(* IEC 61131-3 sources: RL_MAR/experiments/results/ablation/Ablation_no_role_config_deepseek-ai_DeepSeek-V3.2_20260603_074104, 94 files *)

(* ---- hard_92.st ---- *)
FUNCTION_BLOCK FB_BreakerControlSystem
VAR_INPUT
    B10_1_Trip : BOOL;
    B10_1_Close : BOOL;
    B10_2_Trip : BOOL;
    B10_2_Close : BOOL;
    B10_12_Trip : BOOL;
    B10_12_Close : BOOL;
    B54_Trip : BOOL;
    B54_Close : BOOL;
    B55_Trip : BOOL;
    B55_Close : BOOL;
    B56_Trip : BOOL;
    B56_Close : BOOL;
    B57_Trip : BOOL;
    B57_Close : BOOL;
END_VAR

VAR_OUTPUT
    Point_1a : INT;
    Point_2a : INT;
    Point_3a : INT;
    Point_4a : INT;
    B10_1_Opened : BOOL;
    B10_1_Closed : BOOL;
    B10_2_Opened : BOOL;
    B10_2_Closed : BOOL;
    B10_12_Opened : BOOL;
    B10_12_Closed : BOOL;
    B54_Opened : BOOL;
    B54_Closed : BOOL;
    B55_Opened : BOOL;
    B55_Closed : BOOL;
    B56_Opened : BOOL;
    B56_Closed : BOOL;
    B57_Opened : BOOL;
    B57_Closed : BOOL;
END_VAR

VAR
    SEL86_OUT : INT;
    MOVE89_OUT : INT;
    SEL66_OUT : INT;
    MOVE69_OUT : INT;
    SEL96_OUT : INT;
    MOVE99_OUT : INT;
    SEL106_OUT : INT;
    MOVE109_OUT : INT;
END_VAR

// Breaker B10_1 State Transition
IF B10_1_Close THEN
    B10_1_Closed := TRUE;
    B10_1_Opened := FALSE;
ELSIF B10_1_Trip THEN
    B10_1_Closed := FALSE;
    B10_1_Opened := TRUE;
END_IF;

// Breaker B10_2 State Transition
IF B10_2_Close THEN
    B10_2_Closed := TRUE;
    B10_2_Opened := FALSE;
ELSIF B10_2_Trip THEN
    B10_2_Closed := FALSE;
    B10_2_Opened := TRUE;
END_IF;

// Breaker B10_12 State Transition
IF B10_12_Close THEN
    B10_12_Closed := TRUE;
    B10_12_Opened := FALSE;
ELSIF B10_12_Trip THEN
    B10_12_Closed := FALSE;
    B10_12_Opened := TRUE;
END_IF;

// Breaker B54 State Transition
IF B54_Close THEN
    B54_Closed := TRUE;
    B54_Opened := FALSE;
ELSIF B54_Trip THEN
    B54_Closed := FALSE;
    B54_Opened := TRUE;
END_IF;

// Breaker B55 State Transition
IF B55_Close THEN
    B55_Closed := TRUE;
    B55_Opened := FALSE;
ELSIF B55_Trip THEN
    B55_Closed := FALSE;
    B55_Opened := TRUE;
END_IF;

// Breaker B56 State Transition
IF B56_Close THEN
    B56_Closed := TRUE;
    B56_Opened := FALSE;
ELSIF B56_Trip THEN
    B56_Closed := FALSE;
    B56_Opened := TRUE;
END_IF;

// Breaker B57 State Transition
IF B57_Close THEN
    B57_Closed := TRUE;
    B57_Opened := FALSE;
ELSIF B57_Trip THEN
    B57_Closed := FALSE;
    B57_Opened := TRUE;
END_IF;

// Point_1a Calculation
IF B54_Closed AND ((B10_12_Closed AND B10_1_Closed) OR B10_2_Closed) THEN
    Point_1a := 0;
ELSE
    Point_1a := 138;
END_IF;

// Point_2a Calculation
IF B55_Closed AND ((B10_12_Closed AND B10_1_Closed) OR B10_2_Closed) THEN
    Point_2a := 0;
ELSE
    Point_2a := 138;
END_IF;

// Point_3a Calculation
IF B56_Closed AND ((B10_12_Closed AND B10_2_Closed) OR B10_1_Closed) THEN
    Point_3a := 0;
ELSE
    Point_3a := 138;
END_IF;

// Point_4a Calculation
IF B57_Closed AND ((B10_12_Closed AND B10_2_Closed) OR B10_1_Closed) THEN
    Point_4a := 0;
ELSE
    Point_4a := 138;
END_IF;

END_FUNCTION_BLOCK

(* ---- hard_93.st ---- *)
FUNCTION_BLOCK FB_CircuitControl
VAR_INPUT
    Reset_All_CB : BOOL;
    Current_Fault_on_TRSF1 : INT;
    Current_Fault_on_66BUS1 : INT;
END_VAR

VAR_OUTPUT
    Short_Circuit_TRSF1 : BOOL;
    Short_Circuit_66BUS : BOOL;
    Open_CB1_66KV : BOOL;
    Open_CB2_66KV : BOOL;
    Open_CB_TRSF1 : BOOL;
    Open_CB2_22KV : BOOL;
END_VAR

VAR
    Threshold500 : INT := 500;
    Prev_Open_CB2_22KV : BOOL;
    Prev_Open_CB1_66KV : BOOL;
    Prev_Open_CB_TRSF1 : BOOL;
    Temp_Open_CB2_22KV : BOOL;
    Temp_Open_CB1_66KV : BOOL;
    Temp_Open_CB_TRSF1 : BOOL;
END_VAR

(* Short circuit detection *)
Short_Circuit_66BUS := (Current_Fault_on_66BUS1 > Threshold500);
Short_Circuit_TRSF1 := (Current_Fault_on_TRSF1 > Threshold500);

(* Store previous states at the beginning of execution cycle *)
Prev_Open_CB2_22KV := Open_CB2_22KV;
Prev_Open_CB1_66KV := Open_CB1_66KV;
Prev_Open_CB_TRSF1 := Open_CB_TRSF1;

(* Initialize temporary variables with current output states *)
Temp_Open_CB2_22KV := Open_CB2_22KV;
Temp_Open_CB1_66KV := Open_CB1_66KV;
Temp_Open_CB_TRSF1 := Open_CB_TRSF1;

(* Reset handling - overrides all other logic *)
IF Reset_All_CB THEN
    Temp_Open_CB2_22KV := FALSE;
    Temp_Open_CB1_66KV := FALSE;
    Temp_Open_CB_TRSF1 := FALSE;
    Open_CB2_66KV := FALSE;  (* Even though spec says always TRUE, reset should override *)
ELSE
    (* First pass of circuit breaker control logic *)
    (* Open_CB2_22KV first condition *)
    IF (NOT Prev_Open_CB2_22KV) AND
       ((Open_CB1_66KV AND Open_CB_TRSF1) OR Short_Circuit_66BUS) THEN
        Temp_Open_CB2_22KV := TRUE;
    END_IF;

    (* Open_CB1_66KV first condition *)
    IF (NOT Temp_Open_CB2_22KV) AND
       ((Prev_Open_CB1_66KV AND Open_CB_TRSF1) OR Short_Circuit_66BUS) THEN
        Temp_Open_CB1_66KV := TRUE;
    END_IF;

    (* Open_CB_TRSF1 first condition *)
    IF (NOT Temp_Open_CB2_22KV) AND
       ((Open_CB1_66KV AND Prev_Open_CB_TRSF1) OR Short_Circuit_66BUS) THEN
        Temp_Open_CB_TRSF1 := TRUE;
    END_IF;

    (* Open_CB2_66KV always TRUE when not reset *)
    Open_CB2_66KV := TRUE;

    (* Update Open_CB2_22KV again *)
    IF (NOT Prev_Open_CB2_22KV) AND
       ((Open_CB2_66KV AND Temp_Open_CB1_66KV AND Temp_Open_CB_TRSF1) OR Short_Circuit_TRSF1) THEN
        Temp_Open_CB2_22KV := TRUE;
    END_IF;

    (* Update Open_CB1_66KV again *)
    IF (NOT Temp_Open_CB2_22KV) AND
       ((Open_CB2_66KV AND Prev_Open_CB1_66KV AND Temp_Open_CB_TRSF1) OR Short_Circuit_TRSF1) THEN
        Temp_Open_CB1_66KV := TRUE;
    END_IF;

    (* Update Open_CB_TRSF1 again *)
    IF (NOT Temp_Open_CB2_22KV) AND
       ((Open_CB2_66KV AND Temp_Open_CB1_66KV AND Prev_Open_CB_TRSF1) OR Short_Circuit_TRSF1) THEN
        Temp_Open_CB_TRSF1 := TRUE;
    END_IF;
END_IF;

(* Apply temporary states to outputs *)
Open_CB2_22KV := Temp_Open_CB2_22KV;
Open_CB1_66KV := Temp_Open_CB1_66KV;
Open_CB_TRSF1 := Temp_Open_CB_TRSF1;

END_FUNCTION_BLOCK

(* ---- hard_94.st ---- *)
FUNCTION_BLOCK FB_AdvancedCircuitBreakerControl
VAR_INPUT
    S_AL1_P_B1 : BOOL;
    S_AL1_P_B2 : BOOL;
    S_AL1_MCB : BOOL;
    MCB_BUSY : BOOL;
    MCB_ERROR : BOOL;
    S_AL1_MCBR : BOOL;
    MCBR_BUSY : BOOL;
    MCBR_ERROR : BOOL;
    S_AL1_P_B3 : BOOL;
    S_AL1_MCB2 : BOOL;
    S_AL1_MCBR2 : BOOL;
END_VAR

VAR_OUTPUT
    E_AL1_B1 : BOOL;
    PUWS_AL1_B1_PLUS : BOOL;
    PUWS_AL1_B1_RIGHT : BOOL;
    PAS_AL1_PLUS : BOOL;
    PAS_AL1_TURN : BOOL;
END_VAR

VAR
    PPAL1 : BOOL := 1;
    PP0 : BOOL := 1;
    PP1 : BOOL := 0;
    PP2 : BOOL := 0;
    PP3 : BOOL := 0;
    PP4 : BOOL := 0;
    MCB : BOOL := 1;
    PP5 : BOOL := 0;
    PP7 : BOOL := 0;
    PPL3 : BOOL := 0;
    PPL4 : BOOL := 0;
    MCBR : BOOL := 1;
    PPL5 : BOOL := 0;
    PPL7 : BOOL := 0;
    STABLE : BOOL := 0;
    MCB_CONTROL : BOOL;
END_VAR

METHOD MainLogic : BOOL
VAR_INPUT
END_VAR
VAR_OUTPUT
END_VAR
    STABLE := 0;

    WHILE (STABLE = 0) DO
        STABLE := 1;

        // PP0 to PP1
        IF PP0 AND (NOT MCB_CONTROL) AND (NOT PP1) THEN
            PP0 := 0;
            PP1 := 1;
            STABLE := 0;
        END_IF;

        // PP1 to PP2
        IF PP1 AND S_AL1_P_B1 AND (NOT PP2) THEN
            PP1 := 0;
            PP2 := 1;
            STABLE := 0;
        END_IF;

        // PP2 to PP3
        IF PP2 AND S_AL1_P_B2 AND (NOT MCB_CONTROL) AND (NOT PP3) THEN
            PP2 := 0;
            PP3 := 1;
            STABLE := 0;
        END_IF;

        // PP3 to PP4
        IF PP3 AND S_AL1_MCB AND (NOT PP4) AND (NOT PP1) THEN
            PP3 := 0;
            PP4 := 1;
            PP1 := 1;
            STABLE := 0;
        END_IF;

        // PP4 to PP5
        IF PP4 AND MCB AND MCB_BUSY AND (NOT PP5) THEN
            PP4 := 0;
            MCB := 0;
            PP5 := 1;
            STABLE := 0;
        END_IF;

        // PP5 to PP7
        IF PP5 AND S_AL1_MCB2 AND (NOT PP7) AND (NOT MCB) THEN
            PP5 := 0;
            PP7 := 1;
            MCB := 1;
            STABLE := 0;
        END_IF;

        // PP7 to End
        IF PP7 AND S_AL1_P_B3 THEN
            PP7 := 0;
            STABLE := 0;
        END_IF;

        // PP2 to PPL3
        IF PP2 AND S_AL1_P_B2 AND MCB_CONTROL AND (NOT PPL3) AND (NOT PP1) THEN
            PP2 := 0;
            PPL3 := 1;
            PP1 := 1;
            STABLE := 0;
        END_IF;

        // PPL3 to PPL4
        IF PPL3 AND S_AL1_MCBR AND (NOT PPL4) THEN
            PPL3 := 0;
            PPL4 := 1;
            STABLE := 0;
        END_IF;

        // PPL4 to PPL5
        IF PPL4 AND MCBR AND MCBR_BUSY AND (NOT PPL5) THEN
            PPL4 := 0;
            MCBR := 0;
            PPL5 := 1;
            STABLE := 0;
        END_IF;

        // PPL5 to PPL7
        IF PPL5 AND S_AL1_MCBR2 AND (NOT PPL7) AND (NOT MCBR) THEN
            PPL5 := 0;
            PPL7 := 1;
            MCBR := 1;
            STABLE := 0;
        END_IF;

        // PPL7 to End
        IF PPL7 AND S_AL1_P_B3 THEN
            PPL7 := 0;
            STABLE := 0;
        END_IF;
    END_WHILE;

    // Output Control Logic
    IF PP0 OR PP1 THEN
        E_AL1_B1 := 1;
    END_IF;

    IF PP3 THEN
        MCB_CONTROL := 1;
    END_IF;

    IF PPL3 OR PPL4 THEN
        PAS_AL1_PLUS := 1;
        PAS_AL1_TURN := 1;
    END_IF;

    IF PPAL1 OR PP2 THEN
        PUWS_AL1_B1_PLUS := 1;
    END_IF;

    IF PP2 OR PP3 OR PPL3 THEN
        E_AL1_B1 := 0;
    END_IF;

    IF PP0 OR PP3 THEN
        MCB_CONTROL := 0;
    END_IF;

    IF PP0 OR PP3 OR PP4 THEN
        PAS_AL1_PLUS := 0;
        PAS_AL1_TURN := 0;
    END_IF;

    IF PPAL1 OR PP2 THEN
        PUWS_AL1_B1_RIGHT := 0;
    END_IF;

    MainLogic := TRUE;
END_METHOD
END_FUNCTION_BLOCK

(* ---- hf_1.st ---- *)
FUNCTION_BLOCK StackMin
VAR_INPUT
    push : BOOL;
    pop : BOOL;
    reset : BOOL;
END_VAR
VAR_OUTPUT
    error : BOOL;
    status : WORD;
END_VAR
VAR_IN_OUT
    item : INT;
    stack : ARRAY[0..3] OF INT;
END_VAR
VAR
    top : INT := -1;
    i : INT;
    minIndex : INT;
    minValue : INT;
END_VAR

// Reset takes highest priority
IF reset THEN
    top := -1;
    error := FALSE;
    status := 16#0000;
ELSIF push THEN
    // Push operation
    IF top >= 3 THEN
        // Stack is full
        error := TRUE;
        status := 16#8A04;
    ELSE
        // Perform push
        top := top + 1;
        stack[top] := item;
        error := FALSE;
        status := 16#0000;
    END_IF;
ELSIF pop THEN
    // Pop operation (remove minimum value)
    IF top < 0 THEN
        // Stack is empty
        error := TRUE;
        status := 16#8A05;
    ELSE
        // Find minimum value and its index
        minIndex := 0;
        minValue := stack[0];
        FOR i := 1 TO top DO
            IF stack[i] < minValue THEN
                minValue := stack[i];
                minIndex := i;
            END_IF;
        END_FOR;

        // Return minimum value via item
        item := minValue;

        // Shift elements down to remove the minimum
        FOR i := minIndex TO top - 1 DO
            stack[i] := stack[i + 1];
        END_FOR;

        // Clear the last element (optional but clean)
        stack[top] := 0;

        // Update top index
        top := top - 1;

        error := FALSE;
        status := 16#0000;
    END_IF;
ELSE
    // No operation requested
    error := FALSE;
    status := 16#0000;
END_IF;

END_FUNCTION_BLOCK

(* ---- hf_10.st ---- *)
FUNCTION_BLOCK FloatingAverage
VAR_INPUT
    cyclicExecution : BOOL;
    trigger : BOOL;
    value : REAL;
    windowSize : INT;
    reset : BOOL;
END_VAR

VAR_OUTPUT
    average : REAL;
    windowSizeReached : BOOL;
    error : BOOL;
    status : WORD;
END_VAR

VAR
    dataBuffer : ARRAY[1..100] OF REAL; (* Buffer to store the data values *)
    bufferIndex : INT := 1; (* Index to track the current position in the buffer *)
    sum : REAL := 0.0; (* Sum of the data values in the buffer *)
    count : INT := 0; (* Number of valid data points in buffer *)
    triggerPrev : BOOL := FALSE; (* Previous trigger state for edge detection *)
END_VAR

(* Main execution logic *)
IF reset THEN
    (* Reset all internal variables *)
    bufferIndex := 1;
    sum := 0.0;
    count := 0;
    average := 0.0;
    windowSizeReached := FALSE;
    error := FALSE;
    status := 16#0000;

    (* Clear buffer *)
    FOR i := 1 TO 100 DO
        dataBuffer[i] := 0.0;
    END_FOR;

ELSIF windowSize < 1 OR windowSize > 100 THEN
    (* Window size error *)
    error := TRUE;
    status := 16#8200;
    windowSizeReached := FALSE;

ELSE
    (* Check if we should process new data *)
    IF cyclicExecution OR (trigger AND NOT triggerPrev) THEN
        (* Update buffer with new value *)
        dataBuffer[bufferIndex] := value;

        (* Update sum - subtract old value if buffer is full *)
        IF count < windowSize THEN
            sum := sum + value;
            count := count + 1;
        ELSE
            (* Calculate index of oldest value to be replaced *)
            VAR
                oldestIndex : INT;
            END_VAR

            oldestIndex := bufferIndex - windowSize + 1;
            IF oldestIndex < 1 THEN
                oldestIndex := oldestIndex + 100;
            END_IF;

            sum := sum - dataBuffer[oldestIndex] + value;
        END_IF;

        (* Update buffer index with circular buffer logic *)
        bufferIndex := bufferIndex + 1;
        IF bufferIndex > 100 THEN
            bufferIndex := 1;
        END_IF;

        (* Calculate average *)
        IF count > 0 THEN
            average := sum / count;
        ELSE
            average := 0.0;
        END_IF;

        (* Check if window size is reached *)
        windowSizeReached := (count >= windowSize);

        (* Clear error if window size is valid *)
        error := FALSE;
        status := 16#0000;
    END_IF;

    (* Update trigger previous state for edge detection *)
    triggerPrev := trigger;
END_IF;

END_FUNCTION_BLOCK

(* ---- hf_11.st ---- *)
FUNCTION_BLOCK FB_BottleProcessing
VAR_INPUT
    bottleSensor : BOOL;
    cleaningConfirmButton : BOOL;
    fillingConfirmButton : BOOL;
    cappingConfirmButton : BOOL;
    packingConfirmButton : BOOL;
    finishedButton : BOOL;
END_VAR

VAR_OUTPUT
    Pump_Motor : BOOL;
    Filling_Valve : BOOL;
    Capping_Machine : BOOL;
    Packing_Machine : BOOL;
    Completion_Light : BOOL;
END_VAR

VAR
    State : INT := 0; (* 0=Waiting, 1=Cleaning, 2=Filling, 3=Capping, 4=Packing, 5=Completed *)
END_VAR

CASE State OF
    0: (* Waiting *)
        (* State actions *)
        Pump_Motor := FALSE;
        Filling_Valve := FALSE;
        Capping_Machine := FALSE;
        Packing_Machine := FALSE;
        Completion_Light := FALSE;

        (* State transition *)
        IF bottleSensor THEN
            Pump_Motor := TRUE;
            State := 1;
        END_IF;

    1: (* Cleaning *)
        (* State actions *)
        Pump_Motor := TRUE;
        Filling_Valve := FALSE;
        Capping_Machine := FALSE;
        Packing_Machine := FALSE;
        Completion_Light := FALSE;

        (* State transition *)
        IF cleaningConfirmButton THEN
            Pump_Motor := FALSE;
            Filling_Valve := TRUE;
            State := 2;
        END_IF;

    2: (* Filling *)
        (* State actions *)
        Pump_Motor := FALSE;
        Filling_Valve := TRUE;
        Capping_Machine := FALSE;
        Packing_Machine := FALSE;
        Completion_Light := FALSE;

        (* State transition *)
        IF fillingConfirmButton THEN
            Filling_Valve := FALSE;
            Capping_Machine := TRUE;
            State := 3;
        END_IF;

    3: (* Capping *)
        (* State actions *)
        Pump_Motor := FALSE;
        Filling_Valve := FALSE;
        Capping_Machine := TRUE;
        Packing_Machine := FALSE;
        Completion_Light := FALSE;

        (* State transition *)
        IF cappingConfirmButton THEN
            Capping_Machine := FALSE;
            Packing_Machine := TRUE;
            State := 4;
        END_IF;

    4: (* Packing *)
        (* State actions *)
        Pump_Motor := FALSE;
        Filling_Valve := FALSE;
        Capping_Machine := FALSE;
        Packing_Machine := TRUE;
        Completion_Light := FALSE;

        (* State transition *)
        IF packingConfirmButton THEN
            Packing_Machine := FALSE;
            Completion_Light := TRUE;
            State := 5;
        END_IF;

    5: (* Completed *)
        (* State actions *)
        Pump_Motor := FALSE;
        Filling_Valve := FALSE;
        Capping_Machine := FALSE;
        Packing_Machine := FALSE;
        Completion_Light := TRUE;

        (* State transition *)
        IF finishedButton THEN
            Completion_Light := FALSE;
            (* All outputs already FALSE except Completion_Light which was just turned off *)
            State := 0;
        END_IF;

END_CASE;

END_FUNCTION_BLOCK

(* ---- hf_12.st ---- *)
FUNCTION_BLOCK MaterialMixing
VAR_INPUT
    estop : BOOL; (* Emergency Stop Signal, FALSE: Emergency stop triggered, TRUE: No emergency stop triggered *)
    opeMode : BOOL; (* Operation Mode, FALSE: Manual Operation Mode, TRUE: Automatic Operation Mode *)
    valveAStart : BOOL; (* Valve A Start Button *)
    valveBStart : BOOL; (* Valve B Start Button *)
    valveCStart : BOOL; (* Valve C Start Button *)
    valveDStart : BOOL; (* Valve D Start Button *)
    mixMotorStart : BOOL; (* Mixing Motor Start Button *)
    autoStart : BOOL; (* Automatic Start Button *)
    processMode : BOOL; (* Process Mode *)
    levelSensor : INT; (* Liquid Level Sensor, unit cm *)
    mixMotorComplete : BOOL; (* Mixing Complete Signal *)
END_VAR
VAR_OUTPUT
    valveARun : BOOL; (* Valve A Run Command *)
    valveBRun : BOOL; (* Valve B Run Command *)
    valveCRun : BOOL; (* Valve C Run Command *)
    valveDRun : BOOL; (* Valve D Run Command *)
    mixMotorRun : BOOL; (* Mixing Motor Run Command *)
END_VAR
VAR
    previousValveAStart : BOOL := FALSE;
    previousValveBStart : BOOL := FALSE;
    previousValveCStart : BOOL := FALSE;
    previousValveDStart : BOOL := FALSE;
    previousMixMotorStart : BOOL := FALSE;
    previousAutoStart : BOOL := FALSE;
    autoActive : BOOL := FALSE;
    autoStep : INT := 0;
END_VAR

(* Emergency stop has highest priority - when estop is FALSE, stop all equipment *)
IF NOT estop THEN
    valveARun := FALSE;
    valveBRun := FALSE;
    valveCRun := FALSE;
    valveDRun := FALSE;
    mixMotorRun := FALSE;
    autoActive := FALSE;
    autoStep := 0;
ELSE
    (* Automatic Operation Mode *)
    IF opeMode THEN
        (* Manual valve control is disabled in automatic mode *)
        (* Start automatic sequence on rising edge of autoStart button *)
        IF NOT previousAutoStart AND autoStart THEN
            autoActive := TRUE;
            autoStep := 1;
        END_IF;

        (* Execute automatic sequence *)
        IF autoActive THEN
            CASE autoStep OF
                1: (* Step 1: Open Valve A *)
                    valveARun := TRUE;
                    IF levelSensor >= 50 THEN
                        valveARun := FALSE;
                        autoStep := 2;
                    END_IF;

                2: (* Step 2: Open Valve B *)
                    valveBRun := TRUE;
                    IF levelSensor >= 80 THEN
                        valveBRun := FALSE;
                        autoStep := 3;
                    END_IF;

                3: (* Step 3: Check process mode *)
                    IF processMode THEN
                        autoStep := 4; (* Process Mode TRUE: Go to Valve C step *)
                    ELSE
                        autoStep := 5; (* Process Mode FALSE: Skip to mixing motor *)
                    END_IF;

                4: (* Step 4: Open Valve C (only when processMode is TRUE) *)
                    valveCRun := TRUE;
                    IF levelSensor >= 100 THEN
                        valveCRun := FALSE;
                        autoStep := 5;
                    END_IF;

                5: (* Step 5: Start mixing motor *)
                    mixMotorRun := TRUE;
                    IF mixMotorComplete THEN
                        mixMotorRun := FALSE;
                        autoStep := 6;
                    END_IF;

                6: (* Step 6: Open Valve D to deliver mixture *)
                    valveDRun := TRUE;
                    (* Automatic process ends, reset for next cycle *)
                    autoActive := FALSE;
                    autoStep := 0;
            END_CASE;
        END_IF;

    (* Manual Operation Mode *)
    ELSE
        (* Toggle Valve A on rising edge of valveAStart button *)
        IF NOT previousValveAStart AND valveAStart THEN
            valveARun := NOT valveARun;
        END_IF;

        (* Toggle Valve B on rising edge of valveBStart button *)
        IF NOT previousValveBStart AND valveBStart THEN
            valveBRun := NOT valveBRun;
        END_IF;

        (* Toggle Valve C on rising edge of valveCStart button *)
        IF NOT previousValveCStart AND valveCStart THEN
            valveCRun := NOT valveCRun;
        END_IF;

        (* Toggle Valve D on rising edge of valveDStart button *)
        IF NOT previousValveDStart AND valveDStart THEN
            valveDRun := NOT valveDRun;
        END_IF;

        (* Toggle mixing motor on rising edge of mixMotorStart button *)
        IF NOT previousMixMotorStart AND mixMotorStart THEN
            mixMotorRun := NOT mixMotorRun;
        END_IF;
    END_IF;
END_IF;

(* Update previous states for edge detection *)
previousValveAStart := valveAStart;
previousValveBStart := valveBStart;
previousValveCStart := valveCStart;
previousValveDStart := valveDStart;
previousMixMotorStart := mixMotorStart;
previousAutoStart := autoStart;

END_FUNCTION_BLOCK

(* ---- hf_13.st ---- *)
FUNCTION_BLOCK LightsControl
VAR_INPUT
    button1 : BOOL; (* Button 1: Automatic/Manual Mode Select *)
    button2 : BOOL; (* Button 2: Manual Control/Green Light Req *)
    button3 : BOOL; (* Button 3: Manual Control/Red Light Req *)
    CYCLE_TIME : DINT; (* Time elapsed in current cycle (in ms) *)
END_VAR

VAR_OUTPUT
    greenLight : BOOL; (* Green light *)
    redLight : BOOL; (* Red light *)
    yellowLight : BOOL; (* Yellow light *)
END_VAR

VAR
    (* Timers for control *)
    timerAuto : TON;
    timerGreen : TON;
    timerRed : TON;
    timerYellow : TON;

    currentState : INT := 0;
    autoRunTimer : BOOL;

    (* Internal variables for blinking logic *)
    blinkHalfHz : BOOL;
    blinkOneHzGreen : BOOL;
    blinkOneHzYellow : BOOL;
END_VAR

(* Reset manual timers at start of each cycle *)
timerGreen(IN := FALSE, PT := 1000, CYCLE_TIME := CYCLE_TIME);
timerRed(IN := FALSE, PT := 2000, CYCLE_TIME := CYCLE_TIME);
timerYellow(IN := FALSE, PT := 1000, CYCLE_TIME := CYCLE_TIME);

(* Default light states *)
greenLight := FALSE;
redLight := FALSE;
yellowLight := FALSE;

IF NOT button1 THEN (* Manual Mode *)
    (* Reset automatic mode *)
    autoRunTimer := FALSE;
    timerAuto(IN := FALSE, PT := 1000, CYCLE_TIME := CYCLE_TIME);
    currentState := 0;

    (* Manual mode logic *)
    IF NOT button2 AND NOT button3 THEN
        (* Both FALSE: All lights off *)
        greenLight := FALSE;
        redLight := FALSE;
        yellowLight := FALSE;

    ELSIF button2 AND NOT button3 THEN
        (* Green ON, Red blinks at 0.5Hz *)
        greenLight := TRUE;

        (* Create 0.5Hz blink using timerRed with PT=2000ms *)
        timerRed(IN := TRUE, PT := 2000, CYCLE_TIME := CYCLE_TIME);

        (* For 0.5Hz (2000ms period, 1000ms ON, 1000ms OFF):
           Use timerRed.ET to create square wave *)
        IF timerRed.ET < 1000 THEN
            redLight := TRUE;
        ELSE
            redLight := FALSE;
        END_IF;

        yellowLight := FALSE;

    ELSIF NOT button2 AND button3 THEN
        (* Red ON, Yellow blinks at 1Hz *)
        redLight := TRUE;

        (* Create 1Hz blink using timerYellow with PT=1000ms *)
        timerYellow(IN := TRUE, PT := 1000, CYCLE_TIME := CYCLE_TIME);

        (* For 1Hz (1000ms period, 500ms ON, 500ms OFF):
           Use timerYellow.ET to create square wave *)
        IF timerYellow.ET < 500 THEN
            yellowLight := TRUE;
        ELSE
            yellowLight := FALSE;
        END_IF;

        greenLight := FALSE;

    ELSIF button2 AND button3 THEN
        (* Yellow ON, Green blinks at 1Hz *)
        yellowLight := TRUE;

        (* Create 1Hz blink using timerGreen with PT=1000ms *)
        timerGreen(IN := TRUE, PT := 1000, CYCLE_TIME := CYCLE_TIME);

        (* For 1Hz (1000ms period, 500ms ON, 500ms OFF):
           Use timerGreen.ET to create square wave *)
        IF timerGreen.ET < 500 THEN
            greenLight := TRUE;
        ELSE
            greenLight := FALSE;
        END_IF;

        redLight := FALSE;
    END_IF;

ELSE (* Automatic Mode *)
    (* Start automatic timer *)
    autoRunTimer := TRUE;
    timerAuto(IN := autoRunTimer, PT := 1000, CYCLE_TIME := CYCLE_TIME);

    (* State machine for automatic mode *)
    CASE currentState OF
        0: (* State 0: Green light ON for 1 second *)
            greenLight := TRUE;
            redLight := FALSE;
            yellowLight := FALSE;

            IF timerAuto.Q THEN
                (* Move to next state and reset timer *)
                currentState := 1;
                timerAuto(IN := FALSE, PT := 1000, CYCLE_TIME := CYCLE_TIME);
                timerAuto(IN := TRUE, PT := 1000, CYCLE_TIME := CYCLE_TIME);
            END_IF;

        1: (* State 1: Red light ON for 1 second *)
            greenLight := FALSE;
            redLight := TRUE;
            yellowLight := FALSE;

            IF timerAuto.Q THEN
                (* Move to next state and reset timer *)
                currentState := 2;
                timerAuto(IN := FALSE, PT := 1000, CYCLE_TIME := CYCLE_TIME);
                timerAuto(IN := TRUE, PT := 1000, CYCLE_TIME := CYCLE_TIME);
            END_IF;

        2: (* State 2: Yellow light ON for 1 second *)
            greenLight := FALSE;
            redLight := FALSE;
            yellowLight := TRUE;

            IF timerAuto.Q THEN
                (* Return to State 0 and reset timer *)
                currentState := 0;
                timerAuto(IN := FALSE, PT := 1000, CYCLE_TIME := CYCLE_TIME);
                timerAuto(IN := TRUE, PT := 1000, CYCLE_TIME := CYCLE_TIME);
            END_IF;
    END_CASE;
END_IF;

END_FUNCTION_BLOCK

FUNCTION_BLOCK TON
VAR_INPUT
    IN : BOOL;
    PT : DINT;
    CYCLE_TIME : DINT;
END_VAR
VAR_OUTPUT
    Q : BOOL;
    ET : DINT;
END_VAR
VAR
    elapsedTimeInternal : DINT := 0;
    IN_PREV : BOOL := FALSE;
END_VAR

IF IN THEN
    IF NOT IN_PREV THEN
        (* Rising edge detected, reset timer *)
        elapsedTimeInternal := 0;
    END_IF;

    IF elapsedTimeInternal < PT THEN
        (* Timer is running *)
        elapsedTimeInternal := elapsedTimeInternal + CYCLE_TIME;
        Q := FALSE;
    ELSE
        (* Timer has reached preset time *)
        elapsedTimeInternal := PT;
        Q := TRUE;
    END_IF;

    ET := elapsedTimeInternal;
ELSE
    (* Timer is not active *)
    Q := FALSE;
    ET := 0;
    elapsedTimeInternal := 0;
END_IF;

IN_PREV := IN;

END_FUNCTION_BLOCK

(* ---- hf_14.st ---- *)
FUNCTION_BLOCK TruckGarage
VAR_INPUT
    enter_flag : BOOL;
    exit_flag : BOOL;
    VehicleNumber_in : INT;
END_VAR
VAR_OUTPUT
    truck_row : INT;
    truck_col : INT;
    truck_VehicleNumber : INT;
END_VAR
VAR_IN_OUT
    garage : ARRAY[1..3, 1..5] OF STRUCT
        Occupied : BOOL;
        VehicleNumber : INT;
    END_STRUCT;
END_VAR
VAR
    i : INT;
    j : INT;
    space_found : BOOL;
    exit_found : BOOL;
END_VAR

// Initialize output
truck_row := 0;
truck_col := 0;
truck_VehicleNumber := 0;

// Entry logic
IF enter_flag THEN
    space_found := FALSE;

    // Search from last row to first, last column to first
    FOR i := 3 TO 1 BY -1 DO
        FOR j := 5 TO 1 BY -1 DO
            IF NOT garage[i, j].Occupied AND NOT space_found THEN
                // Found empty space
                garage[i, j].Occupied := TRUE;
                garage[i, j].VehicleNumber := VehicleNumber_in;
                space_found := TRUE;
            END_IF
        END_FOR
    END_FOR
END_IF

// Exit logic
IF exit_flag THEN
    exit_found := FALSE;

    // Search from first row to last, first column to last
    FOR i := 1 TO 3 DO
        FOR j := 1 TO 5 DO
            IF garage[i, j].Occupied AND garage[i, j].VehicleNumber = VehicleNumber_in AND NOT exit_found THEN
                // Found vehicle to exit
                truck_row := i;
                truck_col := j;
                truck_VehicleNumber := garage[i, j].VehicleNumber;

                // Clear the parking space
                garage[i, j].Occupied := FALSE;
                garage[i, j].VehicleNumber := 0;
                exit_found := TRUE;
            END_IF
        END_FOR
    END_FOR
END_IF
END_FUNCTION_BLOCK

(* ---- hf_15.st ---- *)
FUNCTION_BLOCK FB_MergeBytes
VAR_INPUT
    byteArray : ARRAY[1..20] OF DINT; (* Byte array to be merged *)
END_VAR
VAR_OUTPUT
    dwordArray : ARRAY[1..10] OF DINT; (* Merged double word array *)
    mergeDwordNum : DINT; (* Actual number of merged double words *)
END_VAR
VAR
    i, j : INT;
    tempDword : DINT;
    byteIndex : INT;
    dwordIndex : INT;
    maxDwords : INT;
END_VAR
VAR CONSTANT
    BYTE_ARRAY_SIZE : DINT := 20; (* Size of the input byte array *)
    DWORD_ARRAY_SIZE : DINT := 10; (* Size of the output DINT array *)
END_VAR

(* Clear output array *)
FOR i := 1 TO DWORD_ARRAY_SIZE DO
    dwordArray[i] := 0;
END_FOR;

mergeDwordNum := 0;

(* Calculate maximum number of complete 4-byte groups in byteArray *)
maxDwords := BYTE_ARRAY_SIZE / 4; (* Integer division automatically truncates remainder *)

(* Limit by dwordArray capacity *)
IF maxDwords > DWORD_ARRAY_SIZE THEN
    maxDwords := DWORD_ARRAY_SIZE;
END_IF;

(* Merge bytes into double words *)
FOR dwordIndex := 1 TO maxDwords DO
    tempDword := 0;
    byteIndex := (dwordIndex - 1) * 4 + 1;

    (* Merge 4 bytes into one double word *)
    FOR j := 0 TO 3 DO
        (* Shift left and OR with current byte *)
        tempDword := tempDword * 256; (* Equivalent to SHL 8 *)
        tempDword := tempDword OR byteArray[byteIndex + j];
    END_FOR;

    dwordArray[dwordIndex] := tempDword;
    mergeDwordNum := mergeDwordNum + 1;
END_FOR;

END_FUNCTION_BLOCK

(* ---- hf_16.st ---- *)
FUNCTION_BLOCK FB_LinearizeValue
VAR_INPUT
    InputValue : REAL;                    // Raw input value for conversion
END_VAR
VAR_OUTPUT
    LinearizedValue : REAL := 0.0;        // Converted output value
    Error : BOOL := FALSE;                // Error status flag
    Status : WORD := 16#0000;             // Operation status code
END_VAR
VAR
    // No additional variables needed
END_VAR

// Main execution logic
IF InputValue < 1200.0 THEN
    // Below minimum range (InputValue < 1200)
    LinearizedValue := 150.0;
    Error := TRUE;
    Status := 16#8001;
ELSIF InputValue >= 1200.0 AND InputValue < 3600.0 THEN
    // Range 1: Input 1200 to 3600 -> Output 150 to 240
    LinearizedValue := 150.0 + (InputValue - 1200.0) * (240.0 - 150.0) / (3600.0 - 1200.0);
    Error := FALSE;
    Status := 16#0000;
ELSIF InputValue >= 3600.0 AND InputValue < 4800.0 THEN
    // Range 2: Input 3600 to 4800 -> Output 240 to 560
    LinearizedValue := 240.0 + (InputValue - 3600.0) * (560.0 - 240.0) / (4800.0 - 3600.0);
    Error := FALSE;
    Status := 16#0000;
ELSIF InputValue >= 4800.0 AND InputValue <= 7000.0 THEN
    // Range 3: Input 4800 to 7000 -> Output 560 to 720
    LinearizedValue := 560.0 + (InputValue - 4800.0) * (720.0 - 560.0) / (7000.0 - 4800.0);
    Error := FALSE;
    Status := 16#0000;
ELSE
    // Above maximum range (InputValue > 7000)
    LinearizedValue := 720.0;
    Error := TRUE;
    Status := 16#8001;
END_IF;

END_FUNCTION_BLOCK

(* ---- hf_17.st ---- *)
FUNCTION_BLOCK FB_WarehouseManagement
VAR_INPUT
    requestIn : BOOL := FALSE;
    requestOut : BOOL := FALSE;
END_VAR

VAR_OUTPUT
    productNum : INT := 0;
    libFreeNum : INT := 9;
    error : BOOL := FALSE;
    status : WORD := 16#0000;
END_VAR

VAR_IN_OUT
    library : ARRAY[1..9] OF BOOL;
END_VAR

VAR
    i : INT;
    found : BOOL;
    initDone : BOOL := FALSE;
    errFull : WORD := 16#8001;
    errEmpty : WORD := 16#8002;
END_VAR

    (* Reset error status at start of each cycle *)
    error := FALSE;
    status := 16#0000;

    (* Initialize library array on first execution *)
    IF NOT initDone THEN
        i := 1;
        WHILE i <= 9 DO
            library[i] := FALSE;
            i := i + 1;
        END_WHILE;
        productNum := 0;
        libFreeNum := 9;
        initDone := TRUE;
    END_IF;

    (* Handle storage request *)
    IF requestIn THEN
        (* Check if storage is full *)
        IF productNum >= 9 THEN
            error := TRUE;
            status := errFull;
        ELSE
            (* Search for free position from highest to lowest index (FILO) *)
            found := FALSE;
            i := 9;
            WHILE i >= 1 AND NOT found DO
                IF NOT library[i] THEN
                    library[i] := TRUE;
                    productNum := productNum + 1;
                    libFreeNum := libFreeNum - 1;
                    found := TRUE;
                END_IF;
                i := i - 1;
            END_WHILE;

            (* If no free position found despite productNum < 9, set error *)
            IF NOT found THEN
                error := TRUE;
                status := errFull;
            END_IF;
        END_IF;
    END_IF;

    (* Handle retrieval request *)
    IF requestOut THEN
        (* Check if storage is empty *)
        IF productNum <= 0 THEN
            error := TRUE;
            status := errEmpty;
        ELSE
            (* Search for occupied position from lowest to highest index (FIFO) *)
            found := FALSE;
            i := 1;
            WHILE i <= 9 AND NOT found DO
                IF library[i] THEN
                    library[i] := FALSE;
                    productNum := productNum - 1;
                    libFreeNum := libFreeNum + 1;
                    found := TRUE;
                END_IF;
                i := i + 1;
            END_WHILE;

            (* If no occupied position found despite productNum > 0, set error *)
            IF NOT found THEN
                error := TRUE;
                status := errEmpty;
            END_IF;
        END_IF;
    END_IF;

    (* Final consistency check *)
    IF (productNum + libFreeNum) <> 9 THEN
        error := TRUE;
        (* Keep existing status if already set, otherwise set to general error *)
        IF status = 16#0000 THEN
            status := 16#8003;
        END_IF;
    END_IF;

END_FUNCTION_BLOCK

(* ---- hf_18.st ---- *)
FUNCTION_BLOCK FB_ColorLightControl
{ S7_Optimized_Access := 'TRUE' }
VAR_INPUT
    controlButton : BOOL; // Push button for sequence control
END_VAR

VAR_OUTPUT
    greenLight : BOOL; // Green light control signal
    redLight : BOOL; // Red light control signal
    yellowLight : BOOL; // Yellow light control signal
END_VAR

VAR
    state : INT := 1; // State machine control variable
    lastControlButton : BOOL := FALSE; // Previous button state
END_VAR

// Edge detection for button press
IF controlButton AND NOT lastControlButton THEN
    // State transition logic
    state := state + 1;
    IF state > 5 THEN
        state := 1;
    END_IF;
END_IF;

// State output logic
CASE state OF
    1: // State 1: Green Only
        greenLight := TRUE;
        redLight := FALSE;
        yellowLight := FALSE;

    2: // State 2: Red Only
        greenLight := FALSE;
        redLight := TRUE;
        yellowLight := FALSE;

    3: // State 3: Yellow Only
        greenLight := FALSE;
        redLight := FALSE;
        yellowLight := TRUE;

    4: // State 4: All Lights On
        greenLight := TRUE;
        redLight := TRUE;
        yellowLight := TRUE;

    5: // State 5: All Lights Off
        greenLight := FALSE;
        redLight := FALSE;
        yellowLight := FALSE;

    ELSE // Default case for safety
        greenLight := FALSE;
        redLight := FALSE;
        yellowLight := FALSE;
        state := 1;
END_CASE;

// Store current button state for next cycle
lastControlButton := controlButton;

END_FUNCTION_BLOCK

(* ---- hf_19.st ---- *)
FUNCTION_BLOCK FB_DatabaseManager
VAR_INPUT
    dataInput : ARRAY[0..5] OF BYTE;
    storeTrigger : BOOL;
    resetTrigger : BOOL;
END_VAR

VAR_OUTPUT
    usedSpace : INT := 0;
    remainingSpace : INT := 20;
    error : BOOL;
    status : WORD;
END_VAR

VAR_IN_OUT
    dataBase : ARRAY[1..20] OF BYTE;
END_VAR

VAR
    i : INT;
    dataLength : INT;
END_VAR

// Main execution logic
IF resetTrigger THEN
    // Reset operation
    FOR i := 1 TO 20 DO
        dataBase[i] := 0;
    END_FOR;

    usedSpace := 0;
    remainingSpace := 20;
    error := FALSE;
    status := 0;

ELSIF storeTrigger THEN
    // Data storage operation
    dataLength := dataInput[0];

    // Length validation
    IF (dataLength <= 0) OR (dataLength > 5) THEN
        error := TRUE;
        status := 16#8001;
    ELSE
        // Space verification
        IF (usedSpace + dataLength) > 20 THEN
            error := TRUE;
            status := 16#8002;
        ELSE
            // Data storage
            FOR i := 1 TO dataLength DO
                dataBase[usedSpace + i] := dataInput[i];
            END_FOR;

            // Update counters and status
            usedSpace := usedSpace + dataLength;
            remainingSpace := 20 - usedSpace;
            error := FALSE;
            status := 0;
        END_IF;
    END_IF;
END_IF;

END_FUNCTION_BLOCK

(* ---- hf_2.st ---- *)
FUNCTION_BLOCK FindMinMaxValues
VAR_INPUT
    values : ARRAY[1..10] OF DINT;
END_VAR
VAR_OUTPUT
    minValue : DINT;
    minValueIndex : DINT;
    maxValue : DINT;
    maxValueIndex : DINT;
END_VAR
VAR
    i : INT;
END_VAR

BEGIN
    // Initialize with first element
    minValue := values[1];
    minValueIndex := 1;
    maxValue := values[1];
    maxValueIndex := 1;

    // Iterate through remaining elements
    FOR i := 2 TO 10 DO
        // Check for minimum value
        IF values[i] < minValue THEN
            minValue := values[i];
            minValueIndex := i;
        END_IF;

        // Check for maximum value
        IF values[i] > maxValue THEN
            maxValue := values[i];
            maxValueIndex := i;
        END_IF;
    END_FOR;
END_FUNCTION_BLOCK

(* ---- hf_20.st ---- *)
FUNCTION_BLOCK FB_ProductionLineControl
VAR_INPUT
    Mode : BOOL; // Manual/Auto mode selection
    ForwardButton : BOOL; // Forward rotation button
    ReverseButton : BOOL; // Reverse rotation button
    SensorA : BOOL; // Sensor A input
    SensorB : BOOL; // Sensor B input
    SensorC : BOOL; // Sensor C input
    ButtonA : BOOL; // Button A input
    ButtonB : BOOL; // Button B input
    ButtonC : BOOL; // Button C input
END_VAR
VAR_OUTPUT
    MotorForward : BOOL; // Motor forward output
    MotorReverse : BOOL; // Motor reverse output
    CompletionLight : BOOL; // Process completion indicator
END_VAR
VAR
    State : INT; // State machine current state
END_VAR

// Main logic
CASE State OF
    0: // Initialization
        MotorForward := FALSE;
        MotorReverse := FALSE;
        CompletionLight := FALSE;
        State := 1;

    1: // Mode selection and manual control / Automatic State 1
        IF NOT Mode THEN // Manual Mode
            // Forward Motion
            IF ForwardButton AND NOT ReverseButton THEN
                MotorForward := TRUE;
                MotorReverse := FALSE;
            // Reverse Motion
            ELSIF ReverseButton AND NOT ForwardButton THEN
                MotorForward := FALSE;
                MotorReverse := TRUE;
            // Stop Condition (both pressed or neither pressed)
            ELSE
                MotorForward := FALSE;
                MotorReverse := FALSE;
            END_IF;
            CompletionLight := FALSE; // Light off in manual mode
        ELSE // Automatic Mode - State 1: Waiting at Station A
            MotorForward := FALSE;
            MotorReverse := FALSE;
            CompletionLight := FALSE;
            IF SensorA THEN
                State := 2; // Transition to Processing at Station A
            END_IF;
        END_IF;

    2: // Automatic Mode - State 2: Processing at Station A
        IF NOT Mode THEN
            State := 1; // Return to manual control if mode changes
        ELSE
            MotorForward := FALSE;
            MotorReverse := FALSE;
            IF ButtonA THEN
                MotorForward := TRUE;
                MotorReverse := FALSE;
                State := 3; // Transition to Moving to Station B
            END_IF;
        END_IF;

    3: // Automatic Mode - State 3: Moving to Station B
        IF NOT Mode THEN
            State := 1;
        ELSE
            MotorReverse := FALSE; // Safety: ensure reverse is off
            IF SensorB THEN
                MotorForward := FALSE;
                State := 4; // Transition to Processing at Station B
            END_IF;
        END_IF;

    4: // Automatic Mode - State 4: Processing at Station B
        IF NOT Mode THEN
            State := 1;
        ELSE
            MotorForward := FALSE;
            MotorReverse := FALSE;
            IF ButtonB THEN
                MotorForward := TRUE;
                MotorReverse := FALSE;
                State := 5; // Transition to Moving to Station C
            END_IF;
        END_IF;

    5: // Automatic Mode - State 5: Moving to Station C
        IF NOT Mode THEN
            State := 1;
        ELSE
            MotorReverse := FALSE; // Safety: ensure reverse is off
            IF SensorC THEN
                MotorForward := FALSE;
                State := 6; // Transition to Processing at Station C
            END_IF;
        END_IF;

    6: // Automatic Mode - State 6: Processing at Station C
        IF NOT Mode THEN
            State := 1;
            CompletionLight := FALSE;
        ELSE
            MotorForward := FALSE;
            MotorReverse := FALSE;
            IF ButtonC THEN
                CompletionLight := TRUE;
                State := 7; // Transition to Cycle Completion
            END_IF;
        END_IF;

    7: // Automatic Mode - State 7: Cycle Completion
        IF NOT Mode THEN
            State := 1;
            CompletionLight := FALSE;
        ELSE
            IF NOT SensorC THEN // Product removal detected
                CompletionLight := FALSE;
                State := 1; // Return to State 1 for next cycle
            END_IF;
        END_IF;

    ELSE
        State := 0; // Fallback to initialization for invalid states
END_CASE;

END_FUNCTION_BLOCK

(* ---- hf_21.st ---- *)
FUNCTION_BLOCK FB_SplitNumber
VAR_INPUT
    InputNumber : INT;
END_VAR

VAR_OUTPUT
    Thousands : INT;
    Hundreds : INT;
    Tens : INT;
    Ones : INT;
    Min : INT;
    error : BOOL;
    status : WORD;
END_VAR

VAR
    tempNumber : INT;
    minValue : INT;
END_VAR

// Input validation
IF (InputNumber < 0) OR (InputNumber > 9999) THEN
    // Error condition
    error := TRUE;
    status := 16#8001;
    Thousands := 0;
    Hundreds := 0;
    Tens := 0;
    Ones := 0;
    Min := 0;
ELSE
    // Valid input - proceed with processing
    error := FALSE;
    status := 16#0000;

    // Digit separation
    Thousands := InputNumber / 1000;
    Hundreds := (InputNumber MOD 1000) / 100;
    Tens := (InputNumber MOD 100) / 10;
    Ones := InputNumber MOD 10;

    // Minimum non-zero digit detection
    minValue := 32767; // Maximum INT value

    // Check Thousands digit
    IF Thousands > 0 THEN
        minValue := minimal(minValue, Thousands);
    END_IF;

    // Check Hundreds digit
    IF Hundreds > 0 THEN
        minValue := minimal(minValue, Hundreds);
    END_IF;

    // Check Tens digit
    IF Tens > 0 THEN
        minValue := minimal(minValue, Tens);
    END_IF;

    // Check Ones digit
    IF Ones > 0 THEN
        minValue := minimal(minValue, Ones);
    END_IF;

    // Set Min output
    IF minValue = 32767 THEN
        // All digits were zero
        Min := 0;
    ELSE
        Min := minValue;
    END_IF;
END_IF;

END_FUNCTION_BLOCK

FUNCTION minimal : INT
VAR_INPUT
    IN1 : INT;
    IN2 : INT;
END_VAR

IF IN1 <= IN2 THEN
    minimal := IN1;
ELSE
    minimal := IN2;
END_IF;
END_FUNCTION

(* ---- hf_3.st ---- *)
FUNCTION_BLOCK MultiPumpCtrl
VAR_INPUT
    mode : BOOL;
    start : BOOL;
    stop : BOOL;
    priorities : ARRAY[1..5] OF INT;
    selections : ARRAY[1..5] OF BOOL;
END_VAR
VAR_OUTPUT
    RunComds : ARRAY[1..5] OF BOOL;
END_VAR
VAR
    i : INT;
    j : INT;
    maxPriority : INT;
    maxIndex : INT;
    runCount : INT;
    usedInAuto : ARRAY[1..5] OF BOOL;
END_VAR

(* Main logic *)
IF stop THEN
    (* Highest priority: stop signal *)
    FOR i := 1 TO 5 DO
        RunComds[i] := FALSE;
    END_FOR;
ELSIF start THEN
    IF NOT mode THEN
        (* Manual mode *)
        FOR i := 1 TO 5 DO
            RunComds[i] := selections[i];
        END_FOR;
    ELSE
        (* Automatic mode - find 3 highest priority pumps *)
        (* Initialize tracking array *)
        FOR i := 1 TO 5 DO
            usedInAuto[i] := FALSE;
        END_FOR;

        runCount := 0;
        WHILE runCount < 3 DO
            maxPriority := -32768; (* Minimum INT value *)
            maxIndex := 1;

            (* Find highest priority pump not yet selected *)
            FOR i := 1 TO 5 DO
                IF (priorities[i] > maxPriority) AND NOT usedInAuto[i] THEN
                    maxPriority := priorities[i];
                    maxIndex := i;
                END_IF;
            END_FOR;

            (* Mark pump as selected *)
            usedInAuto[maxIndex] := TRUE;
            runCount := runCount + 1;
        END_WHILE;

        (* Set run commands based on selected pumps *)
        FOR i := 1 TO 5 DO
            RunComds[i] := usedInAuto[i];
        END_FOR;
    END_IF;
ELSE
    (* start is FALSE - stop all pumps *)
    FOR i := 1 TO 5 DO
        RunComds[i] := FALSE;
    END_FOR;
END_IF;

END_FUNCTION_BLOCK

(* ---- hf_4.st ---- *)
FUNCTION_BLOCK FB_CalculateDayOfYear
VAR_INPUT
    Year : INT;
    Month : INT;
    Day : INT;
END_VAR

VAR_OUTPUT
    DayOfYear : INT;
    error : BOOL;
    status : WORD;
END_VAR

VAR_TEMP
    idx : INT;
    isLeapYear : BOOL;
    maxDay : INT;
END_VAR

VAR
    DaysInMonth : ARRAY[1..12] OF INT := [31, 28, 31, 30, 31, 30, 31, 31, 30, 31, 30, 31];
END_VAR

(* Initialize outputs *)
DayOfYear := 0;
error := FALSE;
status := 0;

(* 1. Month validation (highest priority) *)
IF (Month < 1) OR (Month > 12) THEN
    error := TRUE;
    status := 16#8002;  (* Invalid month *)
    RETURN;
END_IF;

(* 2. Day validation *)
(* First check if day is positive *)
IF Day <= 0 THEN
    error := TRUE;
    status := 16#8003;  (* Invalid day *)
    RETURN;
END_IF;

(* Determine maximum days for the month *)
maxDay := DaysInMonth[Month];

(* Check for February and leap year *)
IF Month = 2 THEN
    (* Leap year calculation *)
    isLeapYear := (((Year MOD 4) = 0) AND ((Year MOD 100) <> 0)) OR ((Year MOD 400) = 0);

    IF isLeapYear THEN
        maxDay := 29;
    ELSE
        maxDay := 28;
    END_IF;
END_IF;

(* Check if day exceeds maximum for the month *)
IF Day > maxDay THEN
    error := TRUE;
    status := 16#8003;  (* Invalid day *)
    RETURN;
END_IF;

(* 3. Year validation (lowest priority) *)
IF (Year < 1000) OR (Year > 3000) THEN
    error := TRUE;
    status := 16#8001;  (* Invalid year *)
    RETURN;
END_IF;

(* All inputs valid - calculate day of year *)
(* Sum days from completed months *)
FOR idx := 1 TO Month-1 DO
    DayOfYear := DayOfYear + DaysInMonth[idx];

    (* Add extra day for February in leap years *)
    IF (idx = 2) THEN
        (* Recalculate leap year for consistency *)
        isLeapYear := (((Year MOD 4) = 0) AND ((Year MOD 100) <> 0)) OR ((Year MOD 400) = 0);
        IF isLeapYear THEN
            DayOfYear := DayOfYear + 1;
        END_IF;
    END_IF;
END_FOR;

(* Add current day *)
DayOfYear := DayOfYear + Day;

END_FUNCTION_BLOCK

(* ---- hf_5.st ---- *)
FUNCTION_BLOCK SelectSort
VAR_INPUT
    exe : BOOL;
    seq : ARRAY[1..100] OF INT;
END_VAR
VAR_OUTPUT
    error : BOOL;
    status : WORD;
END_VAR
VAR
    i : INT;
    j : INT;
    min_idx : INT;
    temp : INT;
    seq_local : ARRAY[1..100] OF INT;
    exe_prev : BOOL;
    sort_successful : BOOL;
END_VAR

(* Initialize outputs *)
error := TRUE;
status := 16#8A01;

(* Rising edge detection for execution trigger *)
IF exe AND NOT exe_prev THEN
    (* Copy input array to local working array *)
    FOR i := 1 TO 100 DO
        seq_local[i] := seq[i];
    END_FOR;

    (* Selection sort algorithm *)
    FOR i := 1 TO 99 DO
        min_idx := i;
        FOR j := i+1 TO 100 DO
            IF seq_local[j] < seq_local[min_idx] THEN
                min_idx := j;
            END_IF;
        END_FOR;

        IF min_idx <> i THEN
            temp := seq_local[i];
            seq_local[i] := seq_local[min_idx];
            seq_local[min_idx] := temp;
        END_IF;
    END_FOR;

    (* Verify sorting result *)
    sort_successful := TRUE;
    FOR i := 1 TO 99 DO
        IF seq_local[i] > seq_local[i+1] THEN
            sort_successful := FALSE;
            EXIT;
        END_IF;
    END_FOR;

    (* Set outputs based on verification *)
    IF sort_successful THEN
        (* Copy sorted array back to output *)
        FOR i := 1 TO 100 DO
            seq[i] := seq_local[i];
        END_FOR;
        error := FALSE;
        status := 16#0000;
    ELSE
        error := TRUE;
        status := 16#8A01;
    END_IF;
END_IF;

(* Store previous execution state *)
exe_prev := exe;
END_FUNCTION_BLOCK

(* ---- hf_6.st ---- *)
FUNCTION_BLOCK RandomNumberGenerator
VAR_INPUT
    minValue : DINT;
    maxValue : DINT;
    randomSeed_in : DINT;
END_VAR

VAR_OUTPUT
    error : BOOL;
    status : WORD;
    randomNumber : DINT;
END_VAR

VAR
    seed : DINT;
END_VAR

// Check if range is valid
IF minValue > maxValue THEN
    error := TRUE;
    status := 16#8200;
    randomNumber := 0;
ELSE
    // Ensure seed is positive using absolute value
    seed := ABS(randomSeed_in);

    // Generate random number within range using modulo arithmetic
    // Use DINT casting to avoid LINT conversion issues
    randomNumber := minValue + DINT_TO_DINT(seed MOD (maxValue - minValue + 1));

    error := FALSE;
    status := 16#0000;
END_IF

(* ---- hf_7.st ---- *)
FUNCTION_BLOCK AnalogConverter
VAR_INPUT
    count : INT;                                (* Number of channels to process (1-10) *)
    analogValues : ARRAY[1..10] OF REAL;        (* Raw ADC values for each channel *)
END_VAR
VAR_OUTPUT
    channel_enable : ARRAY[1..10] OF BOOL;      (* Enable conversion for each channel *)
    channel_hiLIM : ARRAY[1..10] OF REAL;       (* Upper scaling limit *)
    channel_loLIM : ARRAY[1..10] OF REAL;       (* Lower scaling limit *)
    channel_bipolar : ARRAY[1..10] OF BOOL;     (* FALSE=Unipolar, TRUE=Bipolar *)
    channel_measuringMode : ARRAY[1..10] OF INT;(* 0=Non-temp, 1=Std temp, 2=Climatic temp *)
    channel_retVal : ARRAY[1..10] OF WORD;      (* Status/error code for each channel *)
    channel_outputValue : ARRAY[1..10] OF REAL; (* Converted output values *)
END_VAR
VAR
    i : INT;                                    (* Loop counter *)
    normalizedValue : REAL;                     (* Normalized value for scaling *)
END_VAR

(* Process each channel up to specified count *)
FOR i := 1 TO 10 DO
    IF i <= count THEN
        IF channel_enable[i] THEN
            (* Reset status for enabled channels *)
            channel_retVal[i] := 0;

            (* Validate measuring mode *)
            IF (channel_measuringMode[i] < 0) OR (channel_measuringMode[i] > 2) THEN
                channel_retVal[i] := 16#8001;   (* Invalid measuring mode *)
                channel_outputValue[i] := 0.0;
            ELSE
                (* Perform conversion based on measuring mode *)
                CASE channel_measuringMode[i] OF
                    0: (* Non-temperature measurement *)
                        (* Validate scaling limits *)
                        IF channel_hiLIM[i] <= channel_loLIM[i] THEN
                            channel_retVal[i] := 16#8002; (* Invalid limits *)
                            channel_outputValue[i] := 0.0;
                        ELSE
                            (* Perform scaling based on bipolar setting *)
                            IF channel_bipolar[i] THEN
                                (* Bipolar: -27648.0 to 27648.0 maps to loLIM to hiLIM *)
                                normalizedValue := (analogValues[i] + 27648.0) / (2.0 * 27648.0);
                            ELSE
                                (* Unipolar: 0.0 to 27648.0 maps to loLIM to hiLIM *)
                                normalizedValue := analogValues[i] / 27648.0;
                            END_IF;

                            (* Clamp normalized value to 0.0-1.0 range *)
                            IF normalizedValue < 0.0 THEN
                                normalizedValue := 0.0;
                            ELSIF normalizedValue > 1.0 THEN
                                normalizedValue := 1.0;
                            END_IF;

                            (* Apply linear scaling *)
                            channel_outputValue[i] :=
                                channel_loLIM[i] + normalizedValue * (channel_hiLIM[i] - channel_loLIM[i]);
                        END_IF;

                    1: (* Standard temperature measurement *)
                        channel_outputValue[i] := analogValues[i] / 10.0;

                    2: (* Climatic temperature measurement *)
                        channel_outputValue[i] := analogValues[i] / 100.0;
                END_CASE;
            END_IF;
        ELSE
            (* Channel disabled - maintain previous output value *)
            (* Note: channel_retVal remains unchanged for disabled channels *)
        END_IF;
    ELSE
        (* Beyond specified count - clear outputs *)
        channel_outputValue[i] := 0.0;
        channel_retVal[i] := 0;
    END_IF;
END_FOR;
END_FUNCTION_BLOCK

(* ---- hf_8.st ---- *)
FUNCTION_BLOCK FB_HexDigitAnalyzer
VAR_INPUT
    InputNumber: INT;
END_VAR

VAR_OUTPUT
    Thousands: INT;
    Hundreds: INT;
    Tens: INT;
    Ones: INT;
    MinDigit: INT;
    error: BOOL;
    status: WORD;
END_VAR

VAR
    tempMin: INT;
    digit: INT;
END_VAR

METHOD ProcessDigits: BOOL
VAR_INPUT
END_VAR
VAR
    localMin: INT;
END_VAR

    // Initialize local minimum to maximum possible value
    localMin := 32767;

    // Check thousands digit
    digit := Thousands;
    IF digit <> 0 THEN
        IF digit < localMin THEN
            localMin := digit;
        END_IF;
    END_IF;

    // Check hundreds digit
    digit := Hundreds;
    IF digit <> 0 THEN
        IF digit < localMin THEN
            localMin := digit;
        END_IF;
    END_IF;

    // Check tens digit
    digit := Tens;
    IF digit <> 0 THEN
        IF digit < localMin THEN
            localMin := digit;
        END_IF;
    END_IF;

    // Check ones digit
    digit := Ones;
    IF digit <> 0 THEN
        IF digit < localMin THEN
            localMin := digit;
        END_IF;
    END_IF;

    // Set MinDigit
    IF localMin = 32767 THEN
        MinDigit := 0;  // All digits were zero
    ELSE
        MinDigit := localMin;
    END_IF;

    RETURN TRUE;
END_METHOD

// Main execution
IF (InputNumber < 0) OR (InputNumber > 9999) THEN
    // Error condition
    error := TRUE;
    status := 16#8001;
    Thousands := 0;
    Hundreds := 0;
    Tens := 0;
    Ones := 0;
    MinDigit := 0;
ELSE
    // Valid input - process normally
    error := FALSE;
    status := 16#0000;

    // Separate digits
    Thousands := InputNumber / 1000;
    Hundreds := (InputNumber MOD 1000) / 100;
    Tens := (InputNumber MOD 100) / 10;
    Ones := InputNumber MOD 10;

    // Find minimum non-zero digit
    ProcessDigits();
END_IF;

(* ---- hf_9.st ---- *)
FUNCTION_BLOCK FB_ShellSort
VAR_INPUT
    sortDirection : BOOL; // FALSE = ascending, TRUE = descending
    arr : ARRAY[1..1000] OF DINT;
END_VAR

VAR_OUTPUT
    error : BOOL;
    status : WORD;
    sorted_arr : ARRAY[1..1000] OF DINT;
END_VAR

VAR
    i, j, gap : DINT;
    temp : DINT;
    n : DINT := 1000; // Fixed array size
    ascending : BOOL;
END_VAR

// Initialize outputs
error := FALSE;
status := 16#0000;

// Copy input array to output array
FOR i := 1 TO n DO
    sorted_arr[i] := arr[i];
END_FOR;

// Array size validation
IF n <= 1 THEN
    error := TRUE;
    status := 16#8200;
    RETURN;
END_IF;

IF n > 1000 THEN
    error := TRUE;
    status := 16#8201;
    RETURN;
END_IF;

// Determine sort direction
ascending := NOT sortDirection; // FALSE = ascending, TRUE = descending

// Shell Sort implementation
gap := n / 2;
WHILE gap > 0 DO
    FOR i := gap + 1 TO n DO
        temp := sorted_arr[i];
        j := i;

        // Inner loop with direction check
        WHILE (j > gap) AND
              ((ascending AND (sorted_arr[j - gap] > temp)) OR
               (NOT ascending AND (sorted_arr[j - gap] < temp))) DO
            sorted_arr[j] := sorted_arr[j - gap];
            j := j - gap;
        END_WHILE;

        sorted_arr[j] := temp;
    END_FOR;

    gap := gap / 2;
END_WHILE;

// Set success status if no errors occurred
IF NOT error THEN
    status := 16#0000;
END_IF;

(* ---- med_22.st ---- *)
FUNCTION_BLOCK CottonCandyMachine
VAR_INPUT
    SugarLevel : REAL; (* Input for sugar level *)
    SpinningSpeed : INT; (* Input for spinning speed *)
END_VAR
VAR_OUTPUT
    SugarFeeder : BOOL; (* Output to control sugar feeding *)
    MotorSpeed : INT; (* Output to control spinning motor speed *)
END_VAR

// Main logic
IF SugarLevel < 10.0 THEN
    SugarFeeder := TRUE;
ELSE
    SugarFeeder := FALSE;
END_IF;

IF SpinningSpeed > 0 THEN
    MotorSpeed := SpinningSpeed;
ELSE
    MotorSpeed := 0;
END_IF;

END_FUNCTION_BLOCK

(* ---- med_23.st ---- *)
FUNCTION_BLOCK SmartIrrigationSystem
VAR_INPUT
    SoilMoistureSensor1 : REAL;
    SoilMoistureSensor2 : REAL;
    WeatherForecast : INT; (* 0: Sunny, 1: Rainy, 2: Cloudy *)
END_VAR

VAR_OUTPUT
    WaterPump : BOOL;
END_VAR

VAR
    SoilMoistureThreshold : REAL := 30.0;
END_VAR

(* Main logic *)
IF WeatherForecast = 1 THEN
    (* Rainy condition - always turn pump off *)
    WaterPump := FALSE;
ELSIF WeatherForecast = 0 AND
      (SoilMoistureSensor1 < SoilMoistureThreshold OR
       SoilMoistureSensor2 < SoilMoistureThreshold) THEN
    (* Sunny AND at least one sensor below threshold - turn pump on *)
    WaterPump := TRUE;
ELSE
    (* All other conditions - turn pump off *)
    WaterPump := FALSE;
END_IF;

END_FUNCTION_BLOCK

(* ---- med_24.st ---- *)
FUNCTION_BLOCK AutomaticDoorControl
VAR_INPUT
    ProximitySensor : BOOL;
    ElapsedTime : DINT; (* Time in milliseconds since last cycle *)
END_VAR

VAR_OUTPUT
    DoorOpen : BOOL;
END_VAR

VAR
    DoorOpenDuration : DINT := 5000; (* 5 seconds in milliseconds *)
    TimeOpen : DINT := 0; (* Accumulated time door has been open *)
    PreviousSensor : BOOL := FALSE; (* Edge detection for sensor *)
END_VAR

(* Main control logic *)
IF ProximitySensor AND NOT DoorOpen THEN
    (* Open door when sensor activates and door is closed *)
    DoorOpen := TRUE;
    TimeOpen := 0; (* Reset timer *)
ELSIF DoorOpen THEN
    (* Door is currently open *)
    IF ProximitySensor THEN
        (* Sensor still active - keep door open and reset timer *)
        TimeOpen := 0;
    ELSE
        (* Sensor inactive - increment timer *)
        TimeOpen := TimeOpen + ElapsedTime;

        (* Close door if timer exceeds duration *)
        IF TimeOpen >= DoorOpenDuration THEN
            DoorOpen := FALSE;
            TimeOpen := 0; (* Reset for next cycle *)
        END_IF;
    END_IF;
END_IF;

(* Store current sensor state for next cycle *)
PreviousSensor := ProximitySensor;

END_FUNCTION_BLOCK

(* ---- med_25.st ---- *)
FUNCTION_BLOCK WastewaterControl
VAR_INPUT
    InFlow : REAL;
    OutFlow : REAL;
    pH : REAL;
    TankLvl : REAL;
END_VAR

VAR_OUTPUT
    Pump1 : BOOL;
    Pump2 : BOOL;
    Valve1 : BOOL;
    Valve2 : BOOL;
END_VAR

VAR
    LowInFlow : REAL := 100.0;
    HighOutFlow : REAL := 90.0;
    DesiredPH : REAL := 7.0;
    HighTankLvl : REAL := 80.0;
END_VAR

// Main control logic
IF InFlow < LowInFlow THEN
    Pump1 := TRUE;
ELSE
    Pump1 := FALSE;
END_IF;

IF OutFlow > HighOutFlow THEN
    Pump2 := TRUE;
ELSE
    Pump2 := FALSE;
END_IF;

IF pH < DesiredPH THEN
    Valve1 := TRUE;
ELSE
    Valve1 := FALSE;
END_IF;

IF TankLvl > HighTankLvl THEN
    Valve2 := TRUE;
ELSE
    Valve2 := FALSE;
END_IF;

END_FUNCTION_BLOCK

(* ---- med_26.st ---- *)
FUNCTION_BLOCK BookSorting
VAR_INPUT
    RFID1 : BOOL;
    RFID2 : BOOL;
    RFID3 : BOOL;
END_VAR

VAR_OUTPUT
    Motor : BOOL;
    Bin1 : BOOL;
    Bin2 : BOOL;
    Bin3 : BOOL;
END_VAR

// Main logic
Motor := RFID1 OR RFID2 OR RFID3;

Bin1 := RFID1 AND NOT RFID2 AND NOT RFID3;
Bin2 := RFID2 AND NOT RFID1 AND NOT RFID3;
Bin3 := RFID3 AND NOT RFID1 AND NOT RFID2;

END_FUNCTION_BLOCK

(* ---- med_27.st ---- *)
FUNCTION_BLOCK FlowerArrangingMachine
VAR_INPUT
    FlowerTypeSensor : INT; (* Input for detecting flower type *)
    FlowerColorSensor : INT; (* Input for detecting flower color *)
END_VAR
VAR_OUTPUT
    ArrangingMechanism : INT; (* Output for controlling arranging mechanism *)
    ConveyorBelt : BOOL; (* Output for controlling conveyor belt *)
END_VAR

(* Main logic body *)
IF FlowerTypeSensor = 1 AND FlowerColorSensor = 1 THEN
    ArrangingMechanism := 1; (* red type 1 flower *)
ELSIF FlowerTypeSensor = 1 AND FlowerColorSensor = 2 THEN
    ArrangingMechanism := 2; (* blue type 1 flower *)
ELSIF FlowerTypeSensor = 2 AND FlowerColorSensor = 1 THEN
    ArrangingMechanism := 3; (* red type 2 flower *)
ELSIF FlowerTypeSensor = 2 AND FlowerColorSensor = 2 THEN
    ArrangingMechanism := 4; (* blue type 2 flower *)
ELSE
    ArrangingMechanism := 0; (* any other combination *)
END_IF;

(* Control conveyor belt based on arranging mechanism *)
ConveyorBelt := ArrangingMechanism <> 0;

END_FUNCTION_BLOCK

(* ---- med_28.st ---- *)
FUNCTION_BLOCK HomeBrewingSystem
VAR_INPUT
    TemperatureSensor : REAL;     (* Input for temperature measurement *)
    WaterFlowSensor : REAL;       (* Input for water flow measurement *)
    BrewingStartTime : TIME;      (* Input for brewing start time *)
    BrewingDuration : TIME;       (* Input for brewing duration *)
END_VAR
VAR_OUTPUT
    HeatingElement : BOOL;        (* Output for heating element *)
    AgitationMotor : BOOL;        (* Output for agitation motor *)
    HopsDispenser : BOOL;         (* Output for hops dispenser *)
    FermentationTank : BOOL;      (* Output for fermentation tank *)
END_VAR
VAR
    CurrentTime : TIME;           (* Current system time *)
    ElapsedTime : TIME;           (* Time elapsed since brewing start *)
END_VAR

    (* Get current time and calculate elapsed brewing time *)
    CurrentTime := TIME();
    ElapsedTime := CurrentTime - BrewingStartTime;

    (* Control heating element based on temperature *)
    IF TemperatureSensor < 65.0 THEN
        HeatingElement := TRUE;
    ELSE
        HeatingElement := FALSE;
    END_IF;

    (* Control agitation motor based on water flow *)
    IF WaterFlowSensor > 0.5 THEN
        AgitationMotor := TRUE;
    ELSE
        AgitationMotor := FALSE;
    END_IF;

    (* Control hops dispenser - activate after 5 hours of brewing *)
    IF ElapsedTime >= T#5h THEN
        HopsDispenser := TRUE;
    ELSE
        HopsDispenser := FALSE;
    END_IF;

    (* Control fermentation tank - activate after 48 hours of brewing *)
    IF ElapsedTime >= T#48h THEN
        FermentationTank := TRUE;
    ELSE
        FermentationTank := FALSE;
    END_IF;

END_FUNCTION_BLOCK

(* ---- med_29.st ---- *)
FUNCTION_BLOCK DocumentFilingSystem
VAR_INPUT
    DocumentInlet : BOOL; (* Input to detect the arrival of a document *)
    CategorySelector : INT; (* Input to select the document category *)
END_VAR
VAR_OUTPUT
    ConveyorMotor : BOOL; (* Output to control the conveyor motor *)
    StorageBin1 : BOOL; (* Output to activate storage bin 1 *)
    StorageBin2 : BOOL; (* Output to activate storage bin 2 *)
    StorageBin3 : BOOL; (* Output to activate storage bin 3 *)
    StorageBin4 : BOOL; (* Output to activate storage bin 4 *)
END_VAR
VAR
    ValidCategory : BOOL; (* Internal flag for valid category selection *)
END_VAR

(* Determine if category selector is within valid range *)
ValidCategory := (CategorySelector >= 1) AND (CategorySelector <= 4);

(* Main control logic *)
IF DocumentInlet AND ValidCategory THEN
    (* Activate conveyor motor when document is present and category is valid *)
    ConveyorMotor := TRUE;

    (* Activate the appropriate storage bin based on category selection *)
    StorageBin1 := (CategorySelector = 1);
    StorageBin2 := (CategorySelector = 2);
    StorageBin3 := (CategorySelector = 3);
    StorageBin4 := (CategorySelector = 4);
ELSE
    (* Deactivate all outputs when no document or invalid category *)
    ConveyorMotor := FALSE;
    StorageBin1 := FALSE;
    StorageBin2 := FALSE;
    StorageBin3 := FALSE;
    StorageBin4 := FALSE;
END_IF;

END_FUNCTION_BLOCK

(* ---- med_30.st ---- *)
FUNCTION_BLOCK MuseumClimateControl
VAR_INPUT
    HumiditySensor : REAL;
    TemperatureSensor : REAL;
    LightSensor : BOOL;
END_VAR

VAR_OUTPUT
    HVACSystem : BOOL;
    Humidifier : BOOL;
    Dehumidifier : BOOL;
    LightControl : BOOL;
END_VAR

VAR
    TargetHumidity : REAL := 50.0;
    TargetTemperature : REAL := 20.0;
    LightThreshold : BOOL := TRUE;
END_VAR

// Humidity Control Logic
// Activate humidifier when humidity is below target, dehumidifier when above target
// Both off when exactly at target (mutually exclusive)
IF HumiditySensor < TargetHumidity THEN
    Humidifier := TRUE;
    Dehumidifier := FALSE;
ELSIF HumiditySensor > TargetHumidity THEN
    Humidifier := FALSE;
    Dehumidifier := TRUE;
ELSE
    Humidifier := FALSE;
    Dehumidifier := FALSE;
END_IF;

// Temperature Control Logic
// Activate HVAC when temperature is not equal to target (both above and below)
// Turn off when exactly at target temperature
IF TemperatureSensor <> TargetTemperature THEN
    HVACSystem := TRUE;
ELSE
    HVACSystem := FALSE;
END_IF;

// Lighting Control Logic
// Turn off lights when light sensor detects brightness AND threshold is TRUE
// Otherwise keep lights on
IF LightSensor AND LightThreshold THEN
    LightControl := FALSE;
ELSE
    LightControl := TRUE;
END_IF;

END_FUNCTION_BLOCK

(* ---- med_31.st ---- *)
FUNCTION_BLOCK ChargingStationControl
VAR_INPUT
    EVConnected : BOOL;
    EVVoltage : REAL;
    EVCurrent : REAL;
    EVStateOfCharge : REAL;
    ChargingTimer : TIME;
END_VAR

VAR_OUTPUT
    EVCharging : BOOL;
END_VAR

VAR
    VoltageOK : BOOL;
    CurrentOK : BOOL;
    SOCNotFull : BOOL;
    TimerOK : BOOL;
END_VAR

(* Evaluate individual conditions *)
VoltageOK := (EVVoltage > 350.0);
CurrentOK := (EVCurrent <= 32.0);
SOCNotFull := (EVStateOfCharge < 100.0);
TimerOK := (ChargingTimer <= T#2h);

(* Main charging control logic *)
IF EVConnected AND VoltageOK AND CurrentOK AND SOCNotFull AND TimerOK THEN
    EVCharging := TRUE;
ELSE
    EVCharging := FALSE;
END_IF;

END_FUNCTION_BLOCK

(* ---- med_32.st ---- *)
FUNCTION_BLOCK GreenhouseWateringSystem
VAR_INPUT
    SoilMoistureSensor : REAL;   (* Input for soil moisture level (0-100%) *)
    ResponseDelay : TIME := T#5s;  (* Example response delay for the system *)
END_VAR
VAR_OUTPUT
    SprinklersOn : BOOL;         (* Output for controlling sprinklers - on/off *)
END_VAR
VAR
    LastMoistureReading : REAL;
    MoistureThresholdLow : REAL := 30.0;
    MoistureThresholdHigh : REAL := 70.0;
    SystemState : INT := 0;
    DelayTimer : TON;
    DelayElapsed : BOOL;
END_VAR

(* Initialize sprinklers to off state *)
SprinklersOn := FALSE;

(* Store the last moisture reading *)
LastMoistureReading := SoilMoistureSensor;

(* Handle response delay using timer *)
DelayTimer(IN := NOT DelayElapsed, PT := ResponseDelay);
DelayElapsed := DelayTimer.Q;

(* Main control logic - only execute when delay has elapsed *)
IF DelayElapsed THEN
    (* Turn sprinklers ON when moisture is below low threshold *)
    IF SoilMoistureSensor < MoistureThresholdLow THEN
        SprinklersOn := TRUE;
    END_IF;

    (* Turn sprinklers OFF when moisture exceeds high threshold *)
    IF SoilMoistureSensor > MoistureThresholdHigh THEN
        SprinklersOn := FALSE;
    END_IF;

    (* Reset delay timer for next cycle *)
    DelayElapsed := FALSE;
END_IF;

(* State transition logic *)
CASE SystemState OF
    0: (* Initial/Idle state *)
        IF (NOT SprinklersOn) AND (SoilMoistureSensor < MoistureThresholdLow) THEN
            SystemState := 1; (* Transition to activating state *)
        ELSIF SprinklersOn AND (SoilMoistureSensor > MoistureThresholdHigh) THEN
            SystemState := 2; (* Transition to deactivating state *)
        END_IF;

    1: (* Activating state - sprinklers turning on *)
        IF SprinklersOn THEN
            SystemState := 3; (* Transition to active state *)
        END_IF;

    2: (* Deactivating state - sprinklers turning off *)
        IF NOT SprinklersOn THEN
            SystemState := 0; (* Transition back to idle state *)
        END_IF;

    3: (* Active state - sprinklers running *)
        IF SoilMoistureSensor > MoistureThresholdHigh THEN
            SystemState := 2; (* Transition to deactivating state *)
        END_IF;
END_CASE;
END_FUNCTION_BLOCK

(* ---- med_33.st ---- *)
FUNCTION_BLOCK RoboticArmColorSorting
VAR_INPUT
    ColorSensorRed : BOOL;   (* Input: Red color sensor *)
    ColorSensorGreen : BOOL;  (* Input: Green color sensor *)
    ColorSensorBlue : BOOL;   (* Input: Blue color sensor *)
END_VAR

VAR_OUTPUT
    RoboticArmMove : BOOL := FALSE;     (* Output: Control for robotic arm movement *)
    BinRed : BOOL := FALSE;           (* Output: Activate red bin *)
    BinGreen : BOOL := FALSE;         (* Output: Activate green bin *)
    BinBlue : BOOL := FALSE;          (* Output: Activate blue bin *)
END_VAR

(* Internal variables for mutual exclusion logic *)
VAR
    bAnyColorDetected : BOOL;
END_VAR

(* Main logic *)
bAnyColorDetected := ColorSensorRed OR ColorSensorGreen OR ColorSensorBlue;

(* Activate robotic arm when any color is detected *)
RoboticArmMove := bAnyColorDetected;

(* Activate bins with mutual exclusion - only one bin at a time *)
(* Priority: Red > Green > Blue (can be adjusted if needed) *)
IF ColorSensorRed THEN
    BinRed := TRUE;
    BinGreen := FALSE;
    BinBlue := FALSE;
ELSIF ColorSensorGreen THEN
    BinRed := FALSE;
    BinGreen := TRUE;
    BinBlue := FALSE;
ELSIF ColorSensorBlue THEN
    BinRed := FALSE;
    BinGreen := FALSE;
    BinBlue := TRUE;
ELSE
    (* No color detected - deactivate all bins *)
    BinRed := FALSE;
    BinGreen := FALSE;
    BinBlue := FALSE;
END_IF;

END_FUNCTION_BLOCK

(* ---- med_34.st ---- *)
FUNCTION_BLOCK CoffeeMachineControl
VAR_INPUT
    StartButton : BOOL;
    ElapsedTime : DINT; (* Time elapsed since the start of the current process, in milliseconds *)
END_VAR

VAR_OUTPUT
    WaterHeating : BOOL;
    GrinderRunning : BOOL;
    Brewing : BOOL;
    WaterHeated : BOOL;
    GrinderFinished : BOOL;
    CoffeeReady : BOOL;
END_VAR

VAR
    WaterHeatingDuration : DINT := 30000; (* 30 seconds in milliseconds *)
    GrinderDuration : DINT := 15000; (* 15 seconds in milliseconds *)
    BrewingDuration : DINT := 60000; (* 60 seconds in milliseconds *)
    CurrentState : INT := 0; (* 0: Idle, 1: Heating, 2: Grinding, 3: Brewing *)
    ProcessStartTime : DINT := 0;
END_VAR

(* State machine implementation *)
IF NOT StartButton THEN
    (* Reset all outputs and states when start button is not pressed *)
    CurrentState := 0;
    ProcessStartTime := 0;
    WaterHeating := FALSE;
    GrinderRunning := FALSE;
    Brewing := FALSE;
    WaterHeated := FALSE;
    GrinderFinished := FALSE;
    CoffeeReady := FALSE;
ELSE
    CASE CurrentState OF
        0: (* Idle state - waiting for start *)
            WaterHeating := FALSE;
            GrinderRunning := FALSE;
            Brewing := FALSE;
            WaterHeated := FALSE;
            GrinderFinished := FALSE;
            CoffeeReady := FALSE;

            IF StartButton THEN
                (* Start water heating process *)
                CurrentState := 1;
                ProcessStartTime := ElapsedTime;
                WaterHeating := TRUE;
            END_IF;

        1: (* Water heating state *)
            WaterHeating := TRUE;
            GrinderRunning := FALSE;
            Brewing := FALSE;

            IF (ElapsedTime - ProcessStartTime) >= WaterHeatingDuration THEN
                (* Water heating completed *)
                WaterHeating := FALSE;
                WaterHeated := TRUE;
                CurrentState := 2;
                ProcessStartTime := ElapsedTime;
            END_IF;

        2: (* Grinding state *)
            WaterHeating := FALSE;
            GrinderRunning := TRUE;
            Brewing := FALSE;

            IF (ElapsedTime - ProcessStartTime) >= GrinderDuration THEN
                (* Grinding completed *)
                GrinderRunning := FALSE;
                GrinderFinished := TRUE;
                CurrentState := 3;
                ProcessStartTime := ElapsedTime;
            END_IF;

        3: (* Brewing state *)
            WaterHeating := FALSE;
            GrinderRunning := FALSE;
            Brewing := TRUE;

            IF (ElapsedTime - ProcessStartTime) >= BrewingDuration THEN
                (* Brewing completed *)
                Brewing := FALSE;
                CoffeeReady := TRUE;
                CurrentState := 0; (* Return to idle state *)
                ProcessStartTime := 0;
            END_IF;

    END_CASE;
END_IF;

END_FUNCTION_BLOCK

(* ---- med_35.st ---- *)
FUNCTION_BLOCK FB_SimpleCalculation
VAR_INPUT
    INPUT_VAR1 : INT := 2;
    VAR2 : INT := 0;
END_VAR

VAR_OUTPUT
    OUTPUT_VAR1 : INT;
    OUTPUT_VAR2 : INT;
END_VAR

VAR
    COUNTER2 : INT := 0;
    LoopIndex : INT;
END_VAR

// Initialization
OUTPUT_VAR1 := INPUT_VAR1;
OUTPUT_VAR2 := VAR2;

// First loop: Multiply OUTPUT_VAR1 by 2 for 5 iterations
FOR LoopIndex := 1 TO 5 DO
    OUTPUT_VAR1 := OUTPUT_VAR1 * 2;
END_FOR;

// Second loop: Increment OUTPUT_VAR2 by 1 for 5 iterations
// Using WHILE loop with COUNTER2 as specified
COUNTER2 := 0;
WHILE COUNTER2 < 5 DO
    OUTPUT_VAR2 := OUTPUT_VAR2 + 1;
    COUNTER2 := COUNTER2 + 1;
END_WHILE;

END_FUNCTION_BLOCK

(* ---- med_36.st ---- *)
FUNCTION_BLOCK FB_ExpandedPoint
VAR_INPUT
    INPUT_VAR2 : INT;
    INPUT_VAR1_X : INT;
    INPUT_VAR1_Y : INT;
    INPUT_VAR3_X : INT := 1;
    INPUT_VAR3_Y : INT := 2;
END_VAR

VAR_OUTPUT
    OUTPUT_VAR2 : INT;
    OUTPUT_VAR1_X : INT;
    OUTPUT_VAR1_Y : INT;
    OUTPUT_VAR3_X : INT;
    OUTPUT_VAR3_Y : INT;
END_VAR

METHOD Execute : BOOL
VAR_INPUT
END_VAR
VAR_OUTPUT
END_VAR
    // Assign input to output
    OUTPUT_VAR2 := INPUT_VAR2;

    // Set fixed values for OUTPUT_VAR1
    OUTPUT_VAR1_X := 1;
    OUTPUT_VAR1_Y := 2;

    // Set fixed values for OUTPUT_VAR3
    OUTPUT_VAR3_X := 100;
    OUTPUT_VAR3_Y := -7000;

    // Return success
    Execute := TRUE;
END_METHOD

END_FUNCTION_BLOCK

(* ---- med_37.st ---- *)
FUNCTION_BLOCK FB_RealValueAdjuster
VAR_INPUT
    x_in : REAL;
END_VAR
VAR_OUTPUT
    x_out : REAL;
END_VAR
VAR
    x_temp : REAL;
    i_temp : INT;
END_VAR

x_temp := x_in;

(* First condition: check if input is exactly 0.0 *)
IF x_in = 0.0 THEN
    x_temp := x_temp + 1.0;
END_IF;

(* Second condition: check if input is not 0.0 *)
IF x_in <> 0.0 THEN
    x_temp := x_temp + 1.0;
END_IF;

(* Third condition: convert input to integer and check if not zero *)
i_temp := REAL_TO_INT(x_in);
IF i_temp <> 0 THEN
    x_temp := x_temp + 1.0;
END_IF;

x_out := x_temp;

END_FUNCTION_BLOCK

(* ---- med_38.st ---- *)
FUNCTION_BLOCK SolarPanelTracking
VAR_INPUT
    SolarIntensity : REAL;      (* Input: Solar intensity in percentage *)
    CurrentTime : TIME;         (* Input: Current time of day *)
END_VAR

VAR_OUTPUT
    PanelAngle : REAL := 0.0;   (* Output: Panel angle in degrees *)
END_VAR

VAR
    SunriseTime : TIME := T#6H;    (* Sunrise time set to 6 AM *)
    SunsetTime : TIME := T#18H;    (* Sunset time set to 6 PM *)
    NoonTime : TIME := T#12H;      (* Noon time set to 12 PM *)
    MorningAngle : REAL := 30.0;   (* Angle during morning *)
    NoonAngle : REAL := 60.0;      (* Angle during noon *)
    EveningAngle : REAL := 30.0;   (* Angle during evening *)
    State : INT := 1;              (* Current state *)
    NextState : INT := 1;          (* Next state *)
END_VAR

(* State machine execution *)
State := NextState;

CASE State OF
    1: (* Night/Off State *)
        PanelAngle := 0.0;
        IF (CurrentTime >= SunriseTime) AND (CurrentTime < SunsetTime) THEN
            NextState := 2;  (* Transition to daytime active *)
        ELSE
            NextState := 1;  (* Stay in night state *)
        END_IF;

    2: (* Daytime Active State - Decision making state *)
        IF (SolarIntensity >= 90.0) THEN
            NextState := 3;  (* High intensity -> noon angle *)
        ELSIF (CurrentTime < NoonTime) THEN
            NextState := 4;  (* Morning -> morning angle *)
        ELSE
            NextState := 5;  (* Afternoon -> evening angle *)
        END_IF;

    3: (* High Intensity Noon Angle State *)
        PanelAngle := NoonAngle;
        IF (CurrentTime < SunriseTime) OR (CurrentTime >= SunsetTime) THEN
            NextState := 1;  (* Transition to night *)
        ELSIF (SolarIntensity < 90.0) THEN
            NextState := 2;  (* Intensity dropped -> reevaluate *)
        ELSE
            NextState := 3;  (* Stay in high intensity state *)
        END_IF;

    4: (* Morning Angle State *)
        PanelAngle := MorningAngle;
        IF (CurrentTime < SunriseTime) OR (CurrentTime >= SunsetTime) THEN
            NextState := 1;  (* Transition to night *)
        ELSIF (CurrentTime >= NoonTime) OR (SolarIntensity >= 90.0) THEN
            NextState := 2;  (* Time passed noon or high intensity -> reevaluate *)
        ELSE
            NextState := 4;  (* Stay in morning state *)
        END_IF;

    5: (* Evening Angle State *)
        PanelAngle := EveningAngle;
        IF (CurrentTime < SunriseTime) OR (CurrentTime >= SunsetTime) THEN
            NextState := 1;  (* Transition to night *)
        ELSIF (CurrentTime < NoonTime) OR (SolarIntensity >= 90.0) THEN
            NextState := 2;  (* Time before noon or high intensity -> reevaluate *)
        ELSE
            NextState := 5;  (* Stay in evening state *)
        END_IF;

    ELSE  (* Default case for invalid state *)
        NextState := 1;
        PanelAngle := 0.0;
END_CASE;

(* Ensure panel angle stays within 0 to 90 degrees *)
IF PanelAngle < 0.0 THEN
    PanelAngle := 0.0;
ELSIF PanelAngle > 90.0 THEN
    PanelAngle := 90.0;
END_IF;

END_FUNCTION_BLOCK

(* ---- med_39.st ---- *)
FUNCTION_BLOCK WindTurbineControl
VAR_INPUT
    WindSpeedSensor : REAL; (* Input for measuring wind speed *)
    GeneratorSpeedSensor : REAL; (* Input for measuring generator speed *)
END_VAR

VAR_OUTPUT
    BladePitch : INT; (* Output for blade pitch control (degrees) *)
    GeneratorSpeed : REAL; (* Output for generator speed control (RPM) *)
END_VAR

(* Main control logic *)
IF WindSpeedSensor <= 3.0 THEN
    (* Low wind speed category *)
    BladePitch := -5;
    GeneratorSpeed := 500.0;
ELSIF (WindSpeedSensor > 3.0) AND (WindSpeedSensor <= 5.0) THEN
    (* Moderate wind speed category *)
    BladePitch := 0;
    GeneratorSpeed := 800.0;
ELSE
    (* High wind speed category *)
    BladePitch := 5;
    GeneratorSpeed := 1000.0;
END_IF;

END_FUNCTION_BLOCK

(* ---- med_40.st ---- *)
FUNCTION_BLOCK RockClimbingWallControl
VAR_INPUT
    UserWeightSensor : REAL; (* Input for measuring the user's weight *)
    WallDifficultyLevel : INT; (* Input for setting the wall's initial difficulty level *)
    WallHeight : REAL; (* Input for setting the wall's height *)
    RouteSelector : INT; (* Input for selecting a climbing route *)
END_VAR
VAR_OUTPUT
    ClimbingMotorSpeed : REAL; (* Output for controlling the climbing wall motor speed *)
    WallLights : BOOL; (* Output for controlling wall lighting *)
END_VAR

(* Main logic *)
IF UserWeightSensor > 60.0 THEN
    ClimbingMotorSpeed := 1.0;
ELSE
    ClimbingMotorSpeed := 0.8;
END_IF;

CASE RouteSelector OF
    1: WallDifficultyLevel := 1;
    2: WallDifficultyLevel := 2;
    3: WallDifficultyLevel := 3;
    ELSE
        WallDifficultyLevel := 0;
END_CASE;

IF WallHeight > 5.0 THEN
    WallLights := TRUE;
ELSE
    WallLights := FALSE;
END_IF;

END_FUNCTION_BLOCK

(* ---- med_41.st ---- *)
FUNCTION_BLOCK FishTankControl
VAR_INPUT
    OxygenLevel : REAL; (* Input for oxygen level in the tank *)
    WaterTemperature : REAL; (* Input for water temperature *)
    FeedingTime : TIME; (* Time for scheduled feeding *)
    CurrentTime : TIME; (* Current system time *)
END_VAR
VAR_OUTPUT
    OxygenValve : BOOL; (* Output to control oxygen supply *)
    Heater : BOOL; (* Output to control the heater *)
    Feeder : BOOL; (* Output to control the fish feeder *)
END_VAR

// Main logic
IF OxygenLevel < 5.0 THEN
    OxygenValve := TRUE;
ELSE
    OxygenValve := FALSE;
END_IF;

IF WaterTemperature < 25.0 THEN
    Heater := TRUE;
ELSE
    Heater := FALSE;
END_IF;

IF CurrentTime >= FeedingTime THEN
    Feeder := TRUE;
ELSE
    Feeder := FALSE;
END_IF;

END_FUNCTION_BLOCK

(* ---- med_42.st ---- *)
FUNCTION_BLOCK RetractableRoofControl
VAR_INPUT
    RainSensor : BOOL; (* Input to detect rain *)
    WindSensor : BOOL; (* Input to detect wind *)
    TemperatureSensor : REAL; (* Input to measure temperature *)
END_VAR
VAR_OUTPUT
    RoofMotor : BOOL; (* Output to control the roof motor *)
END_VAR

(* Main control logic *)
IF RainSensor AND WindSensor THEN
    RoofMotor := FALSE; (* Close completely *)
ELSIF RainSensor AND (NOT WindSensor) THEN
    RoofMotor := TRUE; (* Partially closed *)
ELSIF (NOT RainSensor) AND (TemperatureSensor < 20.0) THEN
    RoofMotor := TRUE; (* Close slightly *)
ELSIF (NOT RainSensor) AND (TemperatureSensor >= 20.0) THEN
    RoofMotor := FALSE; (* Fully open *)
ELSE
    RoofMotor := FALSE; (* Default safe state *)
END_IF;

END_FUNCTION_BLOCK

(* ---- med_43.st ---- *)
FUNCTION_BLOCK SandwichMaker
VAR_INPUT
    BreadFeeder : BOOL; (* Input: Detects the presence of bread slices *)
    Ingredient1 : BOOL; (* Input: Detects the presence of Ingredient 1 (e.g., cheese) *)
    Ingredient2 : BOOL; (* Input: Detects the presence of Ingredient 2 (e.g., lettuce) *)
    Ingredient3 : BOOL; (* Input: Detects the presence of Ingredient 3 (e.g., tomatoes) *)
    Condiment1 : BOOL; (* Input: Detects the presence of Condiment 1 (e.g., mayo) *)
    Condiment2 : BOOL; (* Input: Detects the presence of Condiment 2 (e.g., mustard) *)
END_VAR
VAR_OUTPUT
    ConveyorMotor : BOOL; (* Output: Controls the conveyor belt motor *)
    AssembleMotor : BOOL; (* Output: Controls the sandwich assembly motor *)
END_VAR
VAR
    SliceCount : INT := 0; (* Counter for bread slices *)
    PrevBreadState : BOOL := FALSE; (* Previous state of BreadFeeder for edge detection *)
END_VAR

(* Conveyor motor control with slice counting *)
IF BreadFeeder THEN
    ConveyorMotor := TRUE;

    (* Increment slice count only on rising edge of BreadFeeder *)
    IF NOT PrevBreadState THEN
        SliceCount := SliceCount + 1;
    END_IF;
ELSE
    ConveyorMotor := FALSE;
END_IF;

(* Update previous bread state for next cycle *)
PrevBreadState := BreadFeeder;

(* Assembly motor control *)
IF (SliceCount >= 2) AND
   Ingredient1 AND Ingredient2 AND Ingredient3 AND
   Condiment1 AND Condiment2 THEN
    AssembleMotor := TRUE;
ELSE
    AssembleMotor := FALSE;
END_IF;

END_FUNCTION_BLOCK

(* ---- med_44.st ---- *)
FUNCTION_BLOCK DroneChargingStation
VAR_INPUT
    Drone1BatteryLevel : INT := 0; (* Battery level of Drone 1 (0-100%) *)
    Drone2BatteryLevel : INT := 0; (* Battery level of Drone 2 (0-100%) *)
    Drone3BatteryLevel : INT := 0; (* Battery level of Drone 3 (0-100%) *)
    ChargingTime : TIME := T#30s; (* Charging time required for each drone *)
END_VAR
VAR_OUTPUT
    Drone1Status : BOOL := FALSE; (* Status of Drone 1 *)
    Drone2Status : BOOL := FALSE; (* Status of Drone 2 *)
    Drone3Status : BOOL := FALSE; (* Status of Drone 3 *)
    ChargingStationStatus : BOOL := FALSE; (* Charging station status *)
    DroneDeployed : BOOL := FALSE; (* Indicates if a drone is deployed *)
END_VAR
VAR
    TimeRemaining : TIME := T#0s; (* Remaining charging time for the current charging operation *)
    ChargingActive : BOOL := FALSE; (* Internal flag for charging operation *)
    ChargingDrone : INT := 0; (* 0=none, 1=drone1, 2=drone2, 3=drone3 *)
END_VAR

(* Main charging logic *)
IF NOT ChargingActive THEN
    (* Charging station is not in use, check for low battery drones *)
    Drone1Status := FALSE;
    Drone2Status := FALSE;
    Drone3Status := FALSE;
    ChargingStationStatus := FALSE;
    ChargingDrone := 0;

    (* Check drones in order for battery below 20% *)
    IF Drone1BatteryLevel < 20 THEN
        Drone1Status := TRUE;
        ChargingActive := TRUE;
        ChargingStationStatus := TRUE;
        TimeRemaining := ChargingTime;
        ChargingDrone := 1;
    ELSIF Drone2BatteryLevel < 20 THEN
        Drone2Status := TRUE;
        ChargingActive := TRUE;
        ChargingStationStatus := TRUE;
        TimeRemaining := ChargingTime;
        ChargingDrone := 2;
    ELSIF Drone3BatteryLevel < 20 THEN
        Drone3Status := TRUE;
        ChargingActive := TRUE;
        ChargingStationStatus := TRUE;
        TimeRemaining := ChargingTime;
        ChargingDrone := 3;
    END_IF;
ELSE
    (* Charging station is in use *)
    ChargingStationStatus := TRUE;

    (* Decrement charging timer *)
    IF TimeRemaining > T#0s THEN
        TimeRemaining := TimeRemaining - T#1ms; (* Decrement by 1 millisecond *)
    END_IF;

    (* Check if charging is complete *)
    IF TimeRemaining <= T#0s THEN
        Drone1Status := FALSE;
        Drone2Status := FALSE;
        Drone3Status := FALSE;
        ChargingStationStatus := FALSE;
        ChargingActive := FALSE;
        ChargingDrone := 0;
        TimeRemaining := T#0s;
    END_IF;
END_IF;

(* Deployment logic based on battery levels *)
IF DroneDeployed THEN
    (* If a drone is deployed, check if any drone battery is critically low *)
    IF (Drone1BatteryLevel < 10) OR (Drone2BatteryLevel < 10) OR (Drone3BatteryLevel < 10) THEN
        DroneDeployed := FALSE; (* Recall the drone *)
    END_IF;
END_IF;

(* Note: DroneDeployed is set to TRUE by external logic when a drone is deployed *)

END_FUNCTION_BLOCK

(* ---- med_45.st ---- *)
FUNCTION_BLOCK AutomatedSmoothieMaker
VAR_INPUT
    BananaAvailable : BOOL;
    BerryMixAvailable : BOOL;
    SpinachAvailable : BOOL;
    YogurtAvailable : BOOL;
    CustomerPreference : INT;
END_VAR

VAR_OUTPUT
    BlenderMotor : BOOL;
    Dispenser : BOOL;
END_VAR

VAR
    RecipeValid : BOOL;
    IngredientsAvailable : BOOL;
    Recipe1Selected : BOOL;
    Recipe2Selected : BOOL;
    Recipe3Selected : BOOL;
END_VAR

(* Determine which recipe is selected based on customer preference *)
Recipe1Selected := (CustomerPreference = 1);
Recipe2Selected := (CustomerPreference = 2);
Recipe3Selected := (CustomerPreference = 3);

(* Validate customer preference *)
RecipeValid := Recipe1Selected OR Recipe2Selected OR Recipe3Selected;

(* Check ingredient availability for the selected recipe *)
IF Recipe1Selected THEN
    IngredientsAvailable := BananaAvailable AND BerryMixAvailable AND YogurtAvailable;
ELSIF Recipe2Selected THEN
    IngredientsAvailable := BerryMixAvailable AND SpinachAvailable AND YogurtAvailable;
ELSIF Recipe3Selected THEN
    IngredientsAvailable := BananaAvailable AND SpinachAvailable AND YogurtAvailable;
ELSE
    IngredientsAvailable := FALSE;
END_IF;

(* Control outputs based on recipe validity and ingredient availability *)
BlenderMotor := RecipeValid AND IngredientsAvailable;
Dispenser := RecipeValid AND IngredientsAvailable;

END_FUNCTION_BLOCK

(* ---- med_46.st ---- *)
FUNCTION_BLOCK PrecisionEngravingMachine
VAR_INPUT
    DesignSelection : INT;
END_VAR
VAR_OUTPUT
    EngravingDepth : REAL;
    EngravingSpeed : REAL;
    ZAxisMotor : BOOL;
    EngravingMotor : BOOL;
END_VAR
VAR
    CalculatedDepth : REAL;
    CalculatedSpeed : REAL;
END_VAR

CASE DesignSelection OF
    1:
        CalculatedSpeed := 10.0;
        CalculatedDepth := 0.1;
        ZAxisMotor := TRUE;
        EngravingMotor := TRUE;
    2:
        CalculatedSpeed := 8.0;
        CalculatedDepth := 0.2;
        ZAxisMotor := TRUE;
        EngravingMotor := TRUE;
    3:
        CalculatedSpeed := 12.0;
        CalculatedDepth := 0.15;
        ZAxisMotor := TRUE;
        EngravingMotor := TRUE;
ELSE
        CalculatedSpeed := 0.0;
        CalculatedDepth := 0.0;
        ZAxisMotor := FALSE;
        EngravingMotor := FALSE;
END_CASE;

EngravingSpeed := CalculatedSpeed;
EngravingDepth := CalculatedDepth;

END_FUNCTION_BLOCK

(* ---- med_47.st ---- *)
FUNCTION_BLOCK WindowCleaningSystem
VAR_INPUT
    StartButton : BOOL;
    EmergencyStop : BOOL;
    UpperLimit : BOOL;
    LowerLimit : BOOL;
END_VAR

VAR_OUTPUT
    ElevatorUp : BOOL;
    ElevatorDown : BOOL;
    RotateClockwise : BOOL;
    WaterPump : BOOL;
END_VAR

VAR
    CleaningInProgress : BOOL;
    StartRisingEdge : BOOL;
    PrevStartButton : BOOL;
    AtUpperLimit : BOOL;
    AtLowerLimit : BOOL;
    ElevatorMoving : BOOL;
END_VAR

    // Detect rising edge of StartButton
    StartRisingEdge := StartButton AND NOT PrevStartButton;
    PrevStartButton := StartButton;

    // Emergency Stop has highest priority
    IF EmergencyStop THEN
        CleaningInProgress := FALSE;
        ElevatorMoving := FALSE;
        AtUpperLimit := FALSE;
        AtLowerLimit := FALSE;
        ElevatorUp := FALSE;
        ElevatorDown := FALSE;
        RotateClockwise := FALSE;
        WaterPump := FALSE;
    ELSE
        // Start cleaning cycle on rising edge when not already in progress
        IF StartRisingEdge AND NOT CleaningInProgress THEN
            CleaningInProgress := TRUE;
            ElevatorMoving := TRUE;
            AtUpperLimit := FALSE;
            AtLowerLimit := FALSE;
        END_IF;

        // Main cleaning cycle logic
        IF CleaningInProgress THEN
            // Detect when upper limit is reached during upward movement
            IF NOT AtUpperLimit AND UpperLimit AND ElevatorUp THEN
                AtUpperLimit := TRUE;
                ElevatorMoving := FALSE;
            END_IF;

            // Control elevator movement direction
            IF NOT AtUpperLimit AND ElevatorMoving THEN
                // Moving up phase
                ElevatorUp := TRUE;
                ElevatorDown := FALSE;
            ELSIF AtUpperLimit AND NOT AtLowerLimit THEN
                // Moving down phase
                ElevatorUp := FALSE;
                ElevatorDown := TRUE;
                ElevatorMoving := TRUE;
            END_IF;

            // Activate cleaning tools when at upper limit and moving down
            IF AtUpperLimit AND NOT AtLowerLimit THEN
                RotateClockwise := TRUE;
                WaterPump := TRUE;
            ELSE
                RotateClockwise := FALSE;
                WaterPump := FALSE;
            END_IF;

            // Detect when lower limit is reached
            IF LowerLimit AND ElevatorDown THEN
                AtLowerLimit := TRUE;
                ElevatorDown := FALSE;
                ElevatorMoving := FALSE;
                CleaningInProgress := FALSE;
                RotateClockwise := FALSE;
                WaterPump := FALSE;
            END_IF;
        ELSE
            // Idle state - all outputs off
            ElevatorUp := FALSE;
            ElevatorDown := FALSE;
            RotateClockwise := FALSE;
            WaterPump := FALSE;
            ElevatorMoving := FALSE;
        END_IF;
    END_IF;
END_FUNCTION_BLOCK

(* ---- med_48.st ---- *)
FUNCTION_BLOCK ChargingStationControl
VAR_INPUT
    EVConnected : BOOL;
    EVVoltage : REAL;
    EVCurrent : REAL;
    EVStateOfCharge : REAL;
    ChargingTimer : TIME;
    MinimumVoltage : REAL;
    MaximumCurrent : REAL;
    MinimumSOC : REAL;
    ChargingVoltage : REAL;
    ChargingCurrent : REAL;
    MaximumChargingTime : TIME;
END_VAR

VAR_OUTPUT
    EVCharging : BOOL;
END_VAR

VAR
    bStartConditionsMet : BOOL;
    bStopConditionsMet : BOOL;
END_VAR

(* Evaluate start conditions - ALL must be TRUE *)
bStartConditionsMet := EVConnected
    AND (EVVoltage > MinimumVoltage)
    AND (EVCurrent <= MaximumCurrent)
    AND (EVStateOfCharge < 100.0)
    AND (ChargingTimer <= MaximumChargingTime);

(* Evaluate stop conditions - ANY can be TRUE *)
bStopConditionsMet := NOT EVConnected
    OR (EVVoltage <= MinimumVoltage)
    OR (EVCurrent > MaximumCurrent)
    OR (EVStateOfCharge >= 100.0)
    OR (ChargingTimer > MaximumChargingTime);

(* Determine charging output *)
IF bStartConditionsMet AND NOT bStopConditionsMet THEN
    EVCharging := TRUE;
ELSE
    EVCharging := FALSE;
END_IF;

END_FUNCTION_BLOCK
